{attribute 'qualified_only'}
{attribute 'to_string'}

TYPE eDataMappingVarNames :
(*
 * Enumeration for mapping every variable in ST_System_Monitor to a fixed
 * monitoring ID.  The hierarchy is fully expanded at every nesting level.
 *
 * Naming convention:
 *   Structs : <topLevel>_<field>_<subField>_..._<leafField>
 *   Arrays  : <path>_<indexName>  where the index names are:
 *               _AVG      (index 0)
 *               _L1       (index 1)
 *               _L2       (index 2)
 *               _L3       (index 3)
 *               _N        (index 4)
 *               _minimum  (index 5)
 *               _maximum  (index 6)
 *   Only electrical measurement arrays are individually expanded:
 *   ar_ActivePower, ar_ReactivePower, ar_ApparentPower,
 *   ar_PhaseVoltage, ar_LineVoltage, ar_Current,
 *   ar_Frequency, ar_THD, ar_PowerFactor.
 *   The aggregate array variable is NOT included; only individual
 *   per-index entries are present (e.g. ar_Current_AVG, ar_Current_L1).
 *
 *)
(	
None													:= 0,
	(*═════════════════════════════════════════════════════════*)
	(*  Safety and System State    *)
	(*═════════════════════════════════════════════════════════*)
	safety_b_SafetyOK                                          , (* BOOL *)
	safety_b_EstopChannelAOK                                   , (* BOOL *)
	safety_b_EstopChannelBOK                                   , (* BOOL *)
	safety_b_InsulationMonitorOK                               , (* BOOL *)
	safety_b_MRCDBOK                                           , (* BOOL *)
	safety_b_InverterDoorOK                                    , (* BOOL *)
	safety_b_ZptOK                                             , (* BOOL *)
	system_b_SMSnumberConfigured                               , (* BOOL *)
	system_b_CustomNameConfigured                              , (* BOOL *)
	system_s_SystemName                                        , (* STRING(20) *)
	system_b_TransportModePending                              , (* BOOL *)
	system_b_DehumModePending                                  , (* BOOL *)
	system_e_State                                             , (* eSystemState *)
	system_e_gridmode                                          , (* eGridmode *)
	system_e_UgridPowermode                                    , (* eUgridPowermode *)
	system_b_StartAllowed                                      , (* BOOL *)
	system_r_CurrentEfficiency                                 , (* REAL *)
	system_r_AvgEfficiency                                     , (* REAL *)
	system_r_RoundtripEfficiency                               , (* REAL *)
	system_DT_SystemTime                                       , (* DT *)
	system_PowerController_r_CurrentAct                        , (* REAL *)
	system_PowerController_r_Sact                              , (* REAL *)
	system_PowerController_r_PAct                              , (* REAL *)
	system_PowerController_r_QAct                              , (* REAL *)
	system_PowerController_r_PhaseVoltageAct                   , (* REAL *)
	system_PowerController_r_PFact                             , (* REAL *)
	system_PowerController_r_FeedInCurrentLimitActual          , (* REAL *)
	system_PowerController_r_SupplyInCurrentLimitActual        , (* REAL *)
	system_PowerController_b_ThrottlingActive                  , (* BOOL *)
	system_PowerController_ui_ThrottlingType                   , (* UINT *)
	system_PowerController_events_b_ReactivePIDError           , (* BOOL *)
	system_PowerController_events_b_ActivePIDError             , (* BOOL *)
	system_PowerController_events_b_FreqShiftPIDError          , (* BOOL *)
	system_GenGridController_b_active                          , (* BOOL *)
	system_GenGridController_b_faultActive                     , (* BOOL *)
	system_GenGridController_b_gensetHot                       , (* BOOL *)
	system_GenGridController_b_gensetStarting                  , (* BOOL *)
	system_GenGridController_b_ModeTransActive                 , (* BOOL *)
	system_GenGridController_b_ModeTransInhibit                , (* BOOL *)
	system_GenGridController_b_ModeChanged                     , (* BOOL *)
	system_GenGridController_b_ShowModeTrans                   , (* BOOL *)
	system_GenGridController_b_extGensetMode                   , (* BOOL *)
	system_GenGridController_b_gensetcontrol                   , (* BOOL *)
	system_GenGridController_e_BreakerMode                     , (* eBreakerOperationMode *)
	system_GenGridController_e_PowerControlMode                , (* ePowerControlMode *)
	system_GenGridController_e_GensetMode                      , (* eGensetMode *)
	system_GenGridController_e_GensetStartStop                 , (* eGensetStartStop *)
	system_GenGridController_e_state                           , (* eGenGridState *)
	system_GenGridController_e_RunCondition                    , (* eRunCondition *)
	system_GenGridController_events_b_InvalidGensetParameters  , (* BOOL *)
	system_GenGridController_events_b_RotationFieldFault       , (* BOOL *)
	system_GenGridController_events_b_CurrentLimitDisconnect   , (* BOOL *)
	system_GenGridController_events_b_CurrentLimitTrip         , (* BOOL *)
	system_GenGridController_events_b_EmstopDisconnect         , (* BOOL *)
	system_GenGridController_events_b_ShutdownDisconnect       , (* BOOL *)
	system_GenGridController_events_b_OverloadTrip             , (* BOOL *)
	system_GenGridController_events_b_OverFreqTrip             , (* BOOL *)
	system_GenGridController_events_b_UnderFreqTrip            , (* BOOL *)
	system_GenGridController_events_b_OverVoltTrip             , (* BOOL *)
	system_GenGridController_events_b_UnderVoltTrip            , (* BOOL *)
	system_GenGridController_events_b_ShutdownTimeOut          , (* BOOL *)
	system_GenGridController_events_b_SynchronisationFault     , (* BOOL *)
	system_GenGridController_events_b_StartupFault             , (* BOOL *)
	system_GenGridController_events_b_WarmupFault              , (* BOOL *)
	system_GenGridController_events_b_GenDownTrip              , (* BOOL *)
	system_GenGridController_events_b_GridLostTrip             , (* BOOL *)
	system_GenGridController_events_b_TransToGenIsoInhibit     , (* BOOL *)
	system_GenGridController_events_b_TransToGenDroopInhibit   , (* BOOL *)
	system_GenGridController_events_b_TransToGenFixInhibit     , (* BOOL *)
	system_GenGridController_events_b_TransFromInputGridAckRQ  , (* BOOL *)
	system_GenGridController_events_b_TransFromInputGenAckRQ   , (* BOOL *)
	system_GenGridController_events_b_StartingInhibit          , (* BOOL *)
	system_events_b_RestartRequiredMachineName                 , (* BOOL *)
	system_events_b_TimeUpdateFailed                           , (* BOOL *)

	(*═════════════════════════════════════════════════════════*)
	(*  Power Conversion Hardware    *)
	(*═════════════════════════════════════════════════════════*)
	powerstack_e_State                                         , (* eStatusPowerStack *)
	powerstack_e_PowerState                                    , (* ePowerstate *)
	powerstack_e_InverterMode                                  , (* eInverterModes *)
	powerstack_e_PowerMode                                     , (* ePowerModes *)
	powerstack_e_ThrottlingStatus                              , (* ePowerModuleThrottlingState *)
	powerstack_r_VoltageDroop                                  , (* REAL *)
	powerstack_r_FrequencyDroop                                , (* REAL *)
	powerstack_r_ACVoltageD7                                   , (* REAL *)
	powerstack_r_FrequencyD7                                   , (* REAL *)
	powerstack_r_ActivePower                                   , (* REAL *)
	powerstack_r_ReactivePower                                 , (* REAL *)
	powerstack_r_Pmin                                          , (* REAL *)
	powerstack_r_Pmax                                          , (* REAL *)
	powerstack_r_QMax                                          , (* REAL *)
	powerstack_r_QMin                                          , (* REAL *)
	powerstack_r_Smax                                          , (* REAL *)
	powerstack_r_ACcurrentLimit                                , (* REAL *)
	powerstack_r_ACcurrentLimitMax                             , (* REAL *)
	powerstack_r_PowerChangeRate                               , (* REAL *)
	powerstack_r_ApparentPower                                 , (* REAL *)
	powerstack_r_CosPhi                                        , (* REAL *)
	powerstack_r_AcCurrent                                     , (* REAL *)
	powerstack_r_DCPower                                       , (* REAL *)
	powerstack_r_DCVoltage                                     , (* REAL *)
	powerstack_r_DCcurrent                                     , (* REAL *)
	powerstack_r_ACVoltageSupply                               , (* REAL *)
	powerstack_r_FrequencySupply                               , (* REAL *)
	powerstack_r_LoadPercent                                   , (* REAL *)
	powerstack_r_RatedCurrent                                  , (* REAL *)
	powerstack_r_RatedPower                                    , (* REAL *)
	powerstack_r_OvercurrentValueAct                           , (* REAL *)
	powerstack_r_OvercurrentValueMax                           , (* REAL *)
	powerstack_r_ThrottlingValueAct                            , (* REAL *)
	powerstack_b_GridTied                                      , (* BOOL *)
	powerstack_b_GridCodeCheckActive                           , (* BOOL *)
	powerstack_b_GridCodeOK                                    , (* BOOL *)
	powerstack_b_GridACdetected                                , (* BOOL *)
	powerstack_b_InverterGridFormingMode                       , (* BOOL *)
	powerstack_b_ACDetected                                    , (* BOOL *)
	powerstack_b_DCDetected                                    , (* BOOL *)
	powerstack_b_InverterRunning                               , (* BOOL *)
	powerstack_b_StartedState                                  , (* BOOL *)
	powerstack_b_ControlEnabled                                , (* BOOL *)
	powerstack_b_EcomodeAvailable                              , (* BOOL *)
	powerstack_b_StartEnabled                                  , (* BOOL *)
	powerstack_r_MaxTemperature                                , (* REAL *)
	powerstack_t_ShiftHoldTimeRemaining                        , (* TIME *)
	powerstack_t_GridCodeReconnectTime                         , (* TIME *)
	powerstack_Events_b_CoolingDerating                        , (* BOOL *)
	powerstack_Events_b_PlimitShiftingActive                   , (* BOOL *)
	powerstack_Events_b_DCdeviationHigh                        , (* BOOL *)
	powerstack_Events_b_TemperatureWarning                     , (* BOOL *)
	powerstack_Events_b_OvercurrentWarning                     , (* BOOL *)
	powerstack_Events_b_UndervoltageWarning                    , (* BOOL *)
	powerstack_Events_b_OvervoltageWarning                     , (* BOOL *)
	powerstack_Events_b_TemperatureDeviationHigh               , (* BOOL *)
	powerstack_Events_b_PlimitShutdownWarning                  , (* BOOL *)
	powerstack_Events_b_MasterWarning                          , (* BOOL *)
	powerstack_Events_b_SlaveWarning                           , (* BOOL *)
	powerstack_Events_b_GridCodeWarning                        , (* BOOL *)
	powerstack_Events_b_UnderFreqFault                         , (* BOOL *)
	powerstack_Events_b_OverFreqFault                          , (* BOOL *)
	powerstack_Events_b_UnderVoltageFault                      , (* BOOL *)
	powerstack_Events_b_OverVoltageFault                       , (* BOOL *)
	powerstack_Events_b_OvercurrentFault                       , (* BOOL *)
	powerstack_Events_b_PlimitShutdown                         , (* BOOL *)
	powerstack_Events_b_TemperatureFault                       , (* BOOL *)
	powerstack_Events_b_MasterFault                            , (* BOOL *)
	powerstack_Events_b_SlaveFault                             , (* BOOL *)
	powerstack_Events_b_NetcontactorFault                      , (* BOOL *)
	powerstack_Events_b_startupTimeOut                         , (* BOOL *)
	powerstack_Events_b_ShutdownTimeOut                        , (* BOOL *)
	powerstack_Events_ui_shutdownRemainingTime                 , (* UINT *)
	powerstack_PowermoduleMaster_b_online                      , (* BOOL *)
	powerstack_PowermoduleMaster_r_ApparentPower               , (* REAL *)
	powerstack_PowermoduleMaster_r_ActivePower                 , (* REAL *)
	powerstack_PowermoduleMaster_r_ReactivePower               , (* REAL *)
	powerstack_PowermoduleMaster_r_ACVoltageD7                 , (* REAL *)
	powerstack_PowermoduleMaster_r_VoltageDroop                , (* REAL *)
	powerstack_PowermoduleMaster_r_ACVoltageSupply             , (* REAL *)
	powerstack_PowermoduleMaster_r_FrequencyD7                 , (* REAL *)
	powerstack_PowermoduleMaster_r_FrequencyDroop              , (* REAL *)
	powerstack_PowermoduleMaster_r_FrequencySupply             , (* REAL *)
	powerstack_PowermoduleMaster_r_CurrentUnbalance            , (* REAL *)
	powerstack_PowermoduleMaster_r_DCPower                     , (* REAL *)
	powerstack_PowermoduleMaster_r_DCVoltage                   , (* REAL *)
	powerstack_PowermoduleMaster_r_DCCurrent                   , (* REAL *)
	powerstack_PowermoduleMaster_r_ACCurrent                   , (* REAL *)
	powerstack_PowermoduleMaster_r_ActiveCurrent               , (* REAL *)
	powerstack_PowermoduleMaster_r_ReactiveCurrent             , (* REAL *)
	powerstack_PowermoduleMaster_r_LoadPercent                 , (* REAL *)
	powerstack_PowermoduleMaster_r_D7SyncError                 , (* REAL *)
	powerstack_PowermoduleMaster_r_Pmin                        , (* REAL *)
	powerstack_PowermoduleMaster_r_Pmax                        , (* REAL *)
	powerstack_PowermoduleMaster_r_QMax                        , (* REAL *)
	powerstack_PowermoduleMaster_r_Qmin                        , (* REAL *)
	powerstack_PowermoduleMaster_r_Pset                        , (* REAL *)
	powerstack_PowermoduleMaster_r_Qset                        , (* REAL *)
	powerstack_PowermoduleMaster_r_ACcurrentLimit              , (* REAL *)
	powerstack_PowermoduleMaster_r_OverCurrentValue            , (* REAL *)
	powerstack_PowermoduleMaster_r_ModulationIndex             , (* REAL *)
	powerstack_PowermoduleMaster_r_TemperatureInverter         , (* REAL *)
	powerstack_PowermoduleMaster_r_TemperatureGridChoke_1      , (* REAL *)
	powerstack_PowermoduleMaster_r_TemperatureGridChoke_2      , (* REAL *)
	powerstack_PowermoduleMaster_r_TemperatureGridChoke_3      , (* REAL *)
	powerstack_PowermoduleMaster_r_TemperatureCMChoke_1        , (* REAL *)
	powerstack_PowermoduleMaster_r_TemperatureCMChoke_2        , (* REAL *)
	powerstack_PowermoduleMaster_r_TemperatureCMChoke_3        , (* REAL *)
	powerstack_PowermoduleMaster_r_TemperatureCMChoke_4        , (* REAL *)
	powerstack_PowermoduleMaster_r_TemperatureMax              , (* REAL *)
	powerstack_PowermoduleMaster_w_TemperatureFaultWord        , (* WORD *)
	powerstack_PowermoduleMaster_w_OperationHours              , (* WORD *)
	powerstack_PowermoduleMaster_e_PowerMode                   , (* ePowerModes *)
	powerstack_PowermoduleMaster_e_InverterMode                , (* eInverterModes *)
	powerstack_PowermoduleMaster_e_Status                      , (* eStatusPowermodule *)
	powerstack_PowermoduleMaster_e_ThrottlingStatus            , (* ePowerModuleThrottlingState *)
	powerstack_PowermoduleMaster_ui_InverterCommStatus         , (* UINT *)
	powerstack_PowermoduleMaster_ui_BuscouplerCommStatus       , (* UINT *)
	powerstack_PowermoduleMaster_b_MccbTripOK                  , (* BOOL *)
	powerstack_PowermoduleMaster_b_MccbUvr24VdcOK              , (* BOOL *)
	powerstack_PowermoduleMaster_b_MccbFb                      , (* BOOL *)
	powerstack_PowermoduleMaster_b_FanFb                       , (* BOOL *)
	powerstack_PowermoduleMaster_b_DCcontactorFb               , (* BOOL *)
	powerstack_PowermoduleMaster_b_PrechargeContactor          , (* BOOL *)
	powerstack_PowermoduleMaster_b_LimiterActive               , (* BOOL *)
	powerstack_PowermoduleMaster_StatusWord_b_ReadyToDCCharge  , (* BOOL *)
	powerstack_PowermoduleMaster_StatusWord_b_ReadyToOperate   , (* BOOL *)
	powerstack_PowermoduleMaster_StatusWord_b_Running          , (* BOOL *)
	powerstack_PowermoduleMaster_StatusWord_b_Fault            , (* BOOL *)
	powerstack_PowermoduleMaster_StatusWord_b_RunEnabled       , (* BOOL *)
	powerstack_PowermoduleMaster_StatusWord_b_QuickstopNotActive, (* BOOL *)
	powerstack_PowermoduleMaster_StatusWord_b_MCCBControlNotOK , (* BOOL *)
	powerstack_PowermoduleMaster_StatusWord_b_Warning          , (* BOOL *)
	powerstack_PowermoduleMaster_StatusWord_b_DCAtReference    , (* BOOL *)
	powerstack_PowermoduleMaster_StatusWord_b_DCAboveLimit     , (* BOOL *)
	powerstack_PowermoduleMaster_StatusWord_b_WatchdogFeedback , (* BOOL *)
	powerstack_PowermoduleMaster_UgridStatusWord_b_ChargeControlActive, (* BOOL *)
	powerstack_PowermoduleMaster_UgridStatusWord_b_InternalChargingSwitchStatus, (* BOOL *)
	powerstack_PowermoduleMaster_UgridStatusWord_b_MCBcontrol  , (* BOOL *)
	powerstack_PowermoduleMaster_UgridStatusWord_b_MCBStatus   , (* BOOL *)
	powerstack_PowermoduleMaster_UgridStatusWord_b_RunEnabled  , (* BOOL *)
	powerstack_PowermoduleMaster_UgridStatusWord_b_DriveReady  , (* BOOL *)
	powerstack_PowermoduleMaster_UgridStatusWord_b_AFEmodeActive, (* BOOL *)
	powerstack_PowermoduleMaster_UgridStatusWord_b_IslandModeActive, (* BOOL *)
	powerstack_PowermoduleMaster_UgridStatusWord_b_MicrogridModeActive, (* BOOL *)
	powerstack_PowermoduleMaster_UgridStatusWord_b_RunRequestActive, (* BOOL *)
	powerstack_PowermoduleMaster_UgridStatusWord_b_DriveInRunState, (* BOOL *)
	powerstack_PowermoduleMaster_UgridStatusWord_b_FaultActive , (* BOOL *)
	powerstack_PowermoduleMaster_UgridStatusWord_b_SynchronizedToD7, (* BOOL *)
	powerstack_PowermoduleMaster_UgridStatusWord_b_D7MeasurementsOK, (* BOOL *)
	powerstack_PowermoduleMaster_GridcodeStatusWord_b_LineVoltTripLimHigh, (* BOOL *)
	powerstack_PowermoduleMaster_GridcodeStatusWord_b_LineVoltTripLimlow, (* BOOL *)
	powerstack_PowermoduleMaster_GridcodeStatusWord_b_LineFreqTripLimHigh, (* BOOL *)
	powerstack_PowermoduleMaster_GridcodeStatusWord_b_LineFreqTripLimLow, (* BOOL *)
	powerstack_PowermoduleMaster_GridcodeStatusWord_b_LineFreqOK, (* BOOL *)
	powerstack_PowermoduleMaster_GridcodeStatusWord_b_LineVoltOK, (* BOOL *)
	powerstack_PowermoduleMaster_GridcodeStatusWord_b_FRTActive, (* BOOL *)
	powerstack_PowermoduleMaster_GridcodeStatusWord_b_GridCodeTripActive, (* BOOL *)
	powerstack_PowermoduleMaster_Events_b_GeneralFaultFlag     , (* BOOL *)
	powerstack_PowermoduleMaster_Events_b_GeneralWarningFlag   , (* BOOL *)
	powerstack_PowermoduleMaster_Events_b_CMSTemperatureRangeWarning, (* BOOL *)
	powerstack_PowermoduleMaster_Events_b_FanStateUnknownWarning, (* BOOL *)
	powerstack_PowermoduleMaster_Events_b_TempThrottlingActive , (* BOOL *)
	powerstack_PowermoduleMaster_Events_b_CurrThrottlingActive , (* BOOL *)
	powerstack_PowermoduleMaster_Events_b_F1OverCurrent        , (* BOOL *)
	powerstack_PowermoduleMaster_Events_b_F2OverVoltage        , (* BOOL *)
	powerstack_PowermoduleMaster_Events_b_F9UnderVoltage       , (* BOOL *)
	powerstack_PowermoduleMaster_Events_b_F91ShortCircuit      , (* BOOL *)
	powerstack_PowermoduleMaster_Events_b_F3EarthFault         , (* BOOL *)
	powerstack_PowermoduleMaster_Events_b_Spare                , (* BOOL *)
	powerstack_PowermoduleMaster_Events_b_F14UnitOverTemperature, (* BOOL *)
	powerstack_PowermoduleMaster_Events_b_F56TemperatureFault  , (* BOOL *)
	powerstack_PowermoduleMaster_Events_b_F10LineSynchFault    , (* BOOL *)
	powerstack_PowermoduleMaster_Events_b_F52KeypadOCCommFault , (* BOOL *)
	powerstack_PowermoduleMaster_Events_b_F53FieldbusFault     , (* BOOL *)
	powerstack_PowermoduleMaster_Events_b_F59SystembusFault    , (* BOOL *)
	powerstack_PowermoduleMaster_Events_b_F54SlotCommunicationFault, (* BOOL *)
	powerstack_PowermoduleMaster_Events_b_F50Meas4mAFault      , (* BOOL *)
	powerstack_PowermoduleMaster_Events_b_F11OutputPhaseFault  , (* BOOL *)
	powerstack_PowermoduleMaster_Events_b_F80ChargeFault       , (* BOOL *)
	powerstack_PowermoduleMaster_Events_b_F51ExternalFault     , (* BOOL *)
	powerstack_PowermoduleMaster_Events_b_F31IGBTFault         , (* BOOL *)
	powerstack_PowermoduleMaster_Events_b_F64MCBstateFault     , (* BOOL *)
	powerstack_PowermoduleMaster_Events_b_WatchdogError        , (* BOOL *)
	powerstack_PowermoduleMaster_Events_b_24VdcUVRFault        , (* BOOL *)
	powerstack_PowermoduleMaster_Events_b_MCCBtrip             , (* BOOL *)
	powerstack_PowermoduleMaster_Events_b_ShutdownTimeOut      , (* BOOL *)
	powerstack_PowermoduleMaster_Events_b_StartUpTimeOut       , (* BOOL *)
	powerstack_PowermoduleMaster_Events_b_CMChokeTemperatureHigh_1  , (* BOOL *)
	powerstack_PowermoduleMaster_Events_b_CMChokeTemperatureHigh_2  , (* BOOL *)
	powerstack_PowermoduleMaster_Events_b_CMChokeTemperatureHigh_3  , (* BOOL *)
	powerstack_PowermoduleMaster_Events_b_CMChokeTemperatureHigh_4  , (* BOOL *)
	powerstack_PowermoduleMaster_Events_b_CMChokeTemperatureTooHigh_1  , (* BOOL *)
	powerstack_PowermoduleMaster_Events_b_CMChokeTemperatureTooHigh_2  , (* BOOL *)
	powerstack_PowermoduleMaster_Events_b_CMChokeTemperatureTooHigh_3  , (* BOOL *)
	powerstack_PowermoduleMaster_Events_b_CMChokeTemperatureTooHigh_4  , (* BOOL *)
	powerstack_PowermoduleMaster_Events_b_GridChokeTemperatureHigh_1  , (* BOOL *)
	powerstack_PowermoduleMaster_Events_b_GridChokeTemperatureHigh_2  , (* BOOL *)
	powerstack_PowermoduleMaster_Events_b_GridChokeTemperatureHigh_3  , (* BOOL *)
	powerstack_PowermoduleMaster_Events_b_GridChokeTemperatureTooHigh_1  , (* BOOL *)
	powerstack_PowermoduleMaster_Events_b_GridChokeTemperatureTooHigh_2  , (* BOOL *)
	powerstack_PowermoduleMaster_Events_b_GridChokeTemperatureTooHigh_3  , (* BOOL *)
	powerstack_PowermoduleMaster_Events_b_inverterTemperatureHigh, (* BOOL *)
	powerstack_PowermoduleMaster_Events_b_PT100Overrange       , (* BOOL *)
	powerstack_PowermoduleMaster_Events_b_PT100Underrange      , (* BOOL *)
	powerstack_PowermoduleMaster_Events_by_PT100ErrorCount     , (* BYTE *)
	powerstack_PowermoduleMaster_controldata_Controlword_b_ChargeDC, (* BOOL *)
	powerstack_PowermoduleMaster_controldata_Controlword_b_run , (* BOOL *)
	powerstack_PowermoduleMaster_controldata_Controlword_b_Reset, (* BOOL *)
	powerstack_PowermoduleMaster_controldata_Controlword_b_FieldbusControlEnable, (* BOOL *)
	powerstack_PowermoduleMaster_controldata_Controlword_b_WatchdogPulse, (* BOOL *)
	powerstack_PowermoduleMaster_controldata_Controlword_b_ParallelAFE, (* BOOL *)
	powerstack_PowermoduleMaster_controldata_Controlword_b_PIDenable, (* BOOL *)
	powerstack_PowermoduleMaster_controldata_Controlword_b_GridCodeEnable, (* BOOL *)
	powerstack_PowermoduleMaster_controldata_Controlword_b_ExtGridcodeTrip, (* BOOL *)
	powerstack_PowermoduleMaster_controldata_ui_ControlwordValue, (* UINT *)
	powerstack_PowermoduleMaster_controldata_i_invertermode    , (* INT *)
	powerstack_PowermoduleMaster_controldata_i_BaseCurrentRef  , (* INT *)
	powerstack_PowermoduleMaster_controldata_i_ReactiveCurrentRef, (* INT *)
	powerstack_PowermoduleMaster_controldata_i_FrequencyDroop  , (* INT *)
	powerstack_PowermoduleMaster_controldata_i_VoltageDroop    , (* INT *)
	powerstack_PowermoduleMaster_controldata_i_FrequencyDroopOffset, (* INT *)
	powerstack_PowermoduleMaster_controldata_i_VoltageCorrection, (* INT *)
	powerstack_PowermoduleMaster_controldata_i_BaseRefRampRate , (* INT *)
	powerstack_PowermoduleMaster_controldata_i_StartPowerMode  , (* INT *)
	powerstack_PowermoduleMaster_controldata_i_StartVoltageMode, (* INT *)
	powerstack_PowermoduleMaster_controldata_i_OutActCurrentLimit, (* INT *)
	powerstack_PowermoduleMaster_controldata_i_InActCurrentLimit, (* INT *)
	powerstack_PowermoduleMaster_controldata_i_DCVramprate     , (* INT *)
	powerstack_PowermoduleSlave_b_online                       , (* BOOL *)
	powerstack_PowermoduleSlave_r_ApparentPower                , (* REAL *)
	powerstack_PowermoduleSlave_r_ActivePower                  , (* REAL *)
	powerstack_PowermoduleSlave_r_ReactivePower                , (* REAL *)
	powerstack_PowermoduleSlave_r_ACVoltageD7                  , (* REAL *)
	powerstack_PowermoduleSlave_r_VoltageDroop                 , (* REAL *)
	powerstack_PowermoduleSlave_r_ACVoltageSupply              , (* REAL *)
	powerstack_PowermoduleSlave_r_FrequencyD7                  , (* REAL *)
	powerstack_PowermoduleSlave_r_FrequencyDroop               , (* REAL *)
	powerstack_PowermoduleSlave_r_FrequencySupply              , (* REAL *)
	powerstack_PowermoduleSlave_r_CurrentUnbalance             , (* REAL *)
	powerstack_PowermoduleSlave_r_DCPower                      , (* REAL *)
	powerstack_PowermoduleSlave_r_DCVoltage                    , (* REAL *)
	powerstack_PowermoduleSlave_r_DCCurrent                    , (* REAL *)
	powerstack_PowermoduleSlave_r_ACCurrent                    , (* REAL *)
	powerstack_PowermoduleSlave_r_ActiveCurrent                , (* REAL *)
	powerstack_PowermoduleSlave_r_ReactiveCurrent              , (* REAL *)
	powerstack_PowermoduleSlave_r_LoadPercent                  , (* REAL *)
	powerstack_PowermoduleSlave_r_D7SyncError                  , (* REAL *)
	powerstack_PowermoduleSlave_r_Pmin                         , (* REAL *)
	powerstack_PowermoduleSlave_r_Pmax                         , (* REAL *)
	powerstack_PowermoduleSlave_r_QMax                         , (* REAL *)
	powerstack_PowermoduleSlave_r_Qmin                         , (* REAL *)
	powerstack_PowermoduleSlave_r_Pset                         , (* REAL *)
	powerstack_PowermoduleSlave_r_Qset                         , (* REAL *)
	powerstack_PowermoduleSlave_r_ACcurrentLimit               , (* REAL *)
	powerstack_PowermoduleSlave_r_OverCurrentValue             , (* REAL *)
	powerstack_PowermoduleSlave_r_ModulationIndex              , (* REAL *)
	powerstack_PowermoduleSlave_r_TemperatureInverter          , (* REAL *)
	powerstack_PowermoduleSlave_r_TemperatureGridChoke_1       , (* REAL *)
	powerstack_PowermoduleSlave_r_TemperatureGridChoke_2       , (* REAL *)
	powerstack_PowermoduleSlave_r_TemperatureGridChoke_3       , (* REAL *)
	powerstack_PowermoduleSlave_r_TemperatureCMChoke_1         , (* REAL *)
	powerstack_PowermoduleSlave_r_TemperatureCMChoke_2         , (* REAL *)
	powerstack_PowermoduleSlave_r_TemperatureCMChoke_3         , (* REAL *)
	powerstack_PowermoduleSlave_r_TemperatureCMChoke_4         , (* REAL *)
	powerstack_PowermoduleSlave_r_TemperatureMax               , (* REAL *)
	powerstack_PowermoduleSlave_w_TemperatureFaultWord         , (* WORD *)
	powerstack_PowermoduleSlave_w_OperationHours               , (* WORD *)
	powerstack_PowermoduleSlave_e_PowerMode                    , (* ePowerModes *)
	powerstack_PowermoduleSlave_e_InverterMode                 , (* eInverterModes *)
	powerstack_PowermoduleSlave_e_Status                       , (* eStatusPowermodule *)
	powerstack_PowermoduleSlave_e_ThrottlingStatus             , (* ePowerModuleThrottlingState *)
	powerstack_PowermoduleSlave_ui_InverterCommStatus          , (* UINT *)
	powerstack_PowermoduleSlave_ui_BuscouplerCommStatus        , (* UINT *)
	powerstack_PowermoduleSlave_b_MccbTripOK                   , (* BOOL *)
	powerstack_PowermoduleSlave_b_MccbUvr24VdcOK               , (* BOOL *)
	powerstack_PowermoduleSlave_b_MccbFb                       , (* BOOL *)
	powerstack_PowermoduleSlave_b_FanFb                        , (* BOOL *)
	powerstack_PowermoduleSlave_b_DCcontactorFb                , (* BOOL *)
	powerstack_PowermoduleSlave_b_PrechargeContactor           , (* BOOL *)
	powerstack_PowermoduleSlave_b_LimiterActive                , (* BOOL *)
	powerstack_PowermoduleSlave_StatusWord_b_ReadyToDCCharge   , (* BOOL *)
	powerstack_PowermoduleSlave_StatusWord_b_ReadyToOperate    , (* BOOL *)
	powerstack_PowermoduleSlave_StatusWord_b_Running           , (* BOOL *)
	powerstack_PowermoduleSlave_StatusWord_b_Fault             , (* BOOL *)
	powerstack_PowermoduleSlave_StatusWord_b_RunEnabled        , (* BOOL *)
	powerstack_PowermoduleSlave_StatusWord_b_QuickstopNotActive, (* BOOL *)
	powerstack_PowermoduleSlave_StatusWord_b_MCCBControlNotOK  , (* BOOL *)
	powerstack_PowermoduleSlave_StatusWord_b_Warning           , (* BOOL *)
	powerstack_PowermoduleSlave_StatusWord_b_DCAtReference     , (* BOOL *)
	powerstack_PowermoduleSlave_StatusWord_b_DCAboveLimit      , (* BOOL *)
	powerstack_PowermoduleSlave_StatusWord_b_WatchdogFeedback  , (* BOOL *)
	powerstack_PowermoduleSlave_UgridStatusWord_b_ChargeControlActive, (* BOOL *)
	powerstack_PowermoduleSlave_UgridStatusWord_b_InternalChargingSwitchStatus, (* BOOL *)
	powerstack_PowermoduleSlave_UgridStatusWord_b_MCBcontrol   , (* BOOL *)
	powerstack_PowermoduleSlave_UgridStatusWord_b_MCBStatus    , (* BOOL *)
	powerstack_PowermoduleSlave_UgridStatusWord_b_RunEnabled   , (* BOOL *)
	powerstack_PowermoduleSlave_UgridStatusWord_b_DriveReady   , (* BOOL *)
	powerstack_PowermoduleSlave_UgridStatusWord_b_AFEmodeActive, (* BOOL *)
	powerstack_PowermoduleSlave_UgridStatusWord_b_IslandModeActive, (* BOOL *)
	powerstack_PowermoduleSlave_UgridStatusWord_b_MicrogridModeActive, (* BOOL *)
	powerstack_PowermoduleSlave_UgridStatusWord_b_RunRequestActive, (* BOOL *)
	powerstack_PowermoduleSlave_UgridStatusWord_b_DriveInRunState, (* BOOL *)
	powerstack_PowermoduleSlave_UgridStatusWord_b_FaultActive  , (* BOOL *)
	powerstack_PowermoduleSlave_UgridStatusWord_b_SynchronizedToD7, (* BOOL *)
	powerstack_PowermoduleSlave_UgridStatusWord_b_D7MeasurementsOK, (* BOOL *)
	powerstack_PowermoduleSlave_GridcodeStatusWord_b_LineVoltTripLimHigh, (* BOOL *)
	powerstack_PowermoduleSlave_GridcodeStatusWord_b_LineVoltTripLimlow, (* BOOL *)
	powerstack_PowermoduleSlave_GridcodeStatusWord_b_LineFreqTripLimHigh, (* BOOL *)
	powerstack_PowermoduleSlave_GridcodeStatusWord_b_LineFreqTripLimLow, (* BOOL *)
	powerstack_PowermoduleSlave_GridcodeStatusWord_b_LineFreqOK, (* BOOL *)
	powerstack_PowermoduleSlave_GridcodeStatusWord_b_LineVoltOK, (* BOOL *)
	powerstack_PowermoduleSlave_GridcodeStatusWord_b_FRTActive , (* BOOL *)
	powerstack_PowermoduleSlave_GridcodeStatusWord_b_GridCodeTripActive, (* BOOL *)
	powerstack_PowermoduleSlave_Events_b_GeneralFaultFlag      , (* BOOL *)
	powerstack_PowermoduleSlave_Events_b_GeneralWarningFlag    , (* BOOL *)
	powerstack_PowermoduleSlave_Events_b_CMSTemperatureRangeWarning, (* BOOL *)
	powerstack_PowermoduleSlave_Events_b_FanStateUnknownWarning, (* BOOL *)
	powerstack_PowermoduleSlave_Events_b_TempThrottlingActive  , (* BOOL *)
	powerstack_PowermoduleSlave_Events_b_CurrThrottlingActive  , (* BOOL *)
	powerstack_PowermoduleSlave_Events_b_F1OverCurrent         , (* BOOL *)
	powerstack_PowermoduleSlave_Events_b_F2OverVoltage         , (* BOOL *)
	powerstack_PowermoduleSlave_Events_b_F9UnderVoltage        , (* BOOL *)
	powerstack_PowermoduleSlave_Events_b_F91ShortCircuit       , (* BOOL *)
	powerstack_PowermoduleSlave_Events_b_F3EarthFault          , (* BOOL *)
	powerstack_PowermoduleSlave_Events_b_Spare                 , (* BOOL *)
	powerstack_PowermoduleSlave_Events_b_F14UnitOverTemperature, (* BOOL *)
	powerstack_PowermoduleSlave_Events_b_F56TemperatureFault   , (* BOOL *)
	powerstack_PowermoduleSlave_Events_b_F10LineSynchFault     , (* BOOL *)
	powerstack_PowermoduleSlave_Events_b_F52KeypadOCCommFault  , (* BOOL *)
	powerstack_PowermoduleSlave_Events_b_F53FieldbusFault      , (* BOOL *)
	powerstack_PowermoduleSlave_Events_b_F59SystembusFault     , (* BOOL *)
	powerstack_PowermoduleSlave_Events_b_F54SlotCommunicationFault, (* BOOL *)
	powerstack_PowermoduleSlave_Events_b_F50Meas4mAFault       , (* BOOL *)
	powerstack_PowermoduleSlave_Events_b_F11OutputPhaseFault   , (* BOOL *)
	powerstack_PowermoduleSlave_Events_b_F80ChargeFault        , (* BOOL *)
	powerstack_PowermoduleSlave_Events_b_F51ExternalFault      , (* BOOL *)
	powerstack_PowermoduleSlave_Events_b_F31IGBTFault          , (* BOOL *)
	powerstack_PowermoduleSlave_Events_b_F64MCBstateFault      , (* BOOL *)
	powerstack_PowermoduleSlave_Events_b_WatchdogError         , (* BOOL *)
	powerstack_PowermoduleSlave_Events_b_24VdcUVRFault         , (* BOOL *)
	powerstack_PowermoduleSlave_Events_b_MCCBtrip              , (* BOOL *)
	powerstack_PowermoduleSlave_Events_b_ShutdownTimeOut       , (* BOOL *)
	powerstack_PowermoduleSlave_Events_b_StartUpTimeOut        , (* BOOL *)
	powerstack_PowermoduleSlave_Events_b_CMChokeTemperatureHigh_1  , (* BOOL *)
	powerstack_PowermoduleSlave_Events_b_CMChokeTemperatureHigh_2  , (* BOOL *)
	powerstack_PowermoduleSlave_Events_b_CMChokeTemperatureHigh_3  , (* BOOL *)
	powerstack_PowermoduleSlave_Events_b_CMChokeTemperatureHigh_4  , (* BOOL *)
	powerstack_PowermoduleSlave_Events_b_CMChokeTemperatureTooHigh_1  , (* BOOL *)
	powerstack_PowermoduleSlave_Events_b_CMChokeTemperatureTooHigh_2  , (* BOOL *)
	powerstack_PowermoduleSlave_Events_b_CMChokeTemperatureTooHigh_3  , (* BOOL *)
	powerstack_PowermoduleSlave_Events_b_CMChokeTemperatureTooHigh_4  , (* BOOL *)
	powerstack_PowermoduleSlave_Events_b_GridChokeTemperatureHigh_1  , (* BOOL *)
	powerstack_PowermoduleSlave_Events_b_GridChokeTemperatureHigh_2  , (* BOOL *)
	powerstack_PowermoduleSlave_Events_b_GridChokeTemperatureHigh_3  , (* BOOL *)
	powerstack_PowermoduleSlave_Events_b_GridChokeTemperatureTooHigh_1  , (* BOOL *)
	powerstack_PowermoduleSlave_Events_b_GridChokeTemperatureTooHigh_2  , (* BOOL *)
	powerstack_PowermoduleSlave_Events_b_GridChokeTemperatureTooHigh_3  , (* BOOL *)
	powerstack_PowermoduleSlave_Events_b_inverterTemperatureHigh, (* BOOL *)
	powerstack_PowermoduleSlave_Events_b_PT100Overrange        , (* BOOL *)
	powerstack_PowermoduleSlave_Events_b_PT100Underrange       , (* BOOL *)
	powerstack_PowermoduleSlave_Events_by_PT100ErrorCount      , (* BYTE *)
	powerstack_PowermoduleSlave_controldata_Controlword_b_ChargeDC, (* BOOL *)
	powerstack_PowermoduleSlave_controldata_Controlword_b_run  , (* BOOL *)
	powerstack_PowermoduleSlave_controldata_Controlword_b_Reset, (* BOOL *)
	powerstack_PowermoduleSlave_controldata_Controlword_b_FieldbusControlEnable, (* BOOL *)
	powerstack_PowermoduleSlave_controldata_Controlword_b_WatchdogPulse, (* BOOL *)
	powerstack_PowermoduleSlave_controldata_Controlword_b_ParallelAFE, (* BOOL *)
	powerstack_PowermoduleSlave_controldata_Controlword_b_PIDenable, (* BOOL *)
	powerstack_PowermoduleSlave_controldata_Controlword_b_GridCodeEnable, (* BOOL *)
	powerstack_PowermoduleSlave_controldata_Controlword_b_ExtGridcodeTrip, (* BOOL *)
	powerstack_PowermoduleSlave_controldata_ui_ControlwordValue, (* UINT *)
	powerstack_PowermoduleSlave_controldata_i_invertermode     , (* INT *)
	powerstack_PowermoduleSlave_controldata_i_BaseCurrentRef   , (* INT *)
	powerstack_PowermoduleSlave_controldata_i_ReactiveCurrentRef, (* INT *)
	powerstack_PowermoduleSlave_controldata_i_FrequencyDroop   , (* INT *)
	powerstack_PowermoduleSlave_controldata_i_VoltageDroop     , (* INT *)
	powerstack_PowermoduleSlave_controldata_i_FrequencyDroopOffset, (* INT *)
	powerstack_PowermoduleSlave_controldata_i_VoltageCorrection, (* INT *)
	powerstack_PowermoduleSlave_controldata_i_BaseRefRampRate  , (* INT *)
	powerstack_PowermoduleSlave_controldata_i_StartPowerMode   , (* INT *)
	powerstack_PowermoduleSlave_controldata_i_StartVoltageMode , (* INT *)
	powerstack_PowermoduleSlave_controldata_i_OutActCurrentLimit, (* INT *)
	powerstack_PowermoduleSlave_controldata_i_InActCurrentLimit, (* INT *)
	powerstack_PowermoduleSlave_controldata_i_DCVramprate      , (* INT *)
	powerstack_Netcontactor_e_NetConState                      , (* eNetcontactorState *)
	powerstack_Netcontactor_b_SyncCloseCommand                 , (* BOOL *)
	powerstack_Netcontactor_b_NetConFb                         , (* BOOL *)
	powerstack_Netcontactor_b_NetcontRightFb                   , (* BOOL *)
	powerstack_Netcontactor_b_NetcontLeftFb                    , (* BOOL *)
	powerstack_Netcontactor_events_b_AMFEnabled                , (* BOOL *)
	powerstack_Netcontactor_events_b_ContactorRightFbFault     , (* BOOL *)
	powerstack_Netcontactor_events_b_ContactorLeftFbFault      , (* BOOL *)
	powerstack_Netcontactor_events_b_ContactorFbTimeout        , (* BOOL *)
	powerstack_Netcontactor_events_b_PhaseRotationFault        , (* BOOL *)
	powerstack_Netcontactor_events_b_IllegalLeftFieldSelected  , (* BOOL *)
	powermonitor_PQMeterReady                                  , (* BOOL *)
	powermonitor_InputField_ar_ApparentPower_AVG               , (* REAL *)
	powermonitor_InputField_ar_ApparentPower_L1                , (* REAL *)
	powermonitor_InputField_ar_ApparentPower_L2                , (* REAL *)
	powermonitor_InputField_ar_ApparentPower_L3                , (* REAL *)
	powermonitor_InputField_ar_ReactivePower_AVG               , (* REAL *)
	powermonitor_InputField_ar_ReactivePower_L1                , (* REAL *)
	powermonitor_InputField_ar_ReactivePower_L2                , (* REAL *)
	powermonitor_InputField_ar_ReactivePower_L3                , (* REAL *)
	powermonitor_InputField_ar_ActivePower_AVG                 , (* REAL *)
	powermonitor_InputField_ar_ActivePower_L1                  , (* REAL *)
	powermonitor_InputField_ar_ActivePower_L2                  , (* REAL *)
	powermonitor_InputField_ar_ActivePower_L3                  , (* REAL *)
	powermonitor_InputField_r_EnergyConsumed                   , (* REAL *)
	powermonitor_InputField_r_EnergySupplied                   , (* REAL *)
	powermonitor_InputField_ar_THD_AVG                         , (* REAL *)
	powermonitor_InputField_ar_THD_L1                          , (* REAL *)
	powermonitor_InputField_ar_THD_L2                          , (* REAL *)
	powermonitor_InputField_ar_THD_L3                          , (* REAL *)
	powermonitor_InputField_ar_PowerFactor_AVG                 , (* REAL *)
	powermonitor_InputField_ar_PowerFactor_L1                  , (* REAL *)
	powermonitor_InputField_ar_PowerFactor_L2                  , (* REAL *)
	powermonitor_InputField_ar_PowerFactor_L3                  , (* REAL *)
	powermonitor_InputField_ar_Current_AVG                     , (* REAL *)
	powermonitor_InputField_ar_Current_L1                      , (* REAL *)
	powermonitor_InputField_ar_Current_L2                      , (* REAL *)
	powermonitor_InputField_ar_Current_L3                      , (* REAL *)
	powermonitor_InputField_ar_Current_N                       , (* REAL *)
	powermonitor_InputField_r_CurrentUnbalance                 , (* REAL *)
	powermonitor_InputField_e_ACrotationStatus                 , (* eACRotationState *)
	powermonitor_InputField_ar_PhaseVoltage_AVG                , (* REAL *)
	powermonitor_InputField_ar_PhaseVoltage_L1                 , (* REAL *)
	powermonitor_InputField_ar_PhaseVoltage_L2                 , (* REAL *)
	powermonitor_InputField_ar_PhaseVoltage_L3                 , (* REAL *)
	powermonitor_InputField_ar_LineVoltage_AVG                 , (* REAL *)
	powermonitor_InputField_ar_LineVoltage_L1                  , (* REAL *)
	powermonitor_InputField_ar_LineVoltage_L2                  , (* REAL *)
	powermonitor_InputField_ar_LineVoltage_L3                  , (* REAL *)
	powermonitor_InputField_li_TimeVoltZeroCrossup             , (* LINT *)
	powermonitor_InputField_ar_Frequency_AVG                   , (* REAL *)
	powermonitor_InputField_ar_Frequency_L1                    , (* REAL *)
	powermonitor_InputField_ar_Frequency_L2                    , (* REAL *)
	powermonitor_InputField_ar_Frequency_L3                    , (* REAL *)
	powermonitor_InputField_r_VoltageUnbalance                 , (* REAL *)
	powermonitor_InputField_r_loadshare                        , (* REAL *)
	powermonitor_InputField_Powerlock_1_ar_ApparentPower_AVG    , (* REAL *)
	powermonitor_InputField_Powerlock_2_ar_ApparentPower_AVG    , (* REAL *)
	powermonitor_InputField_Powerlock_1_ar_ApparentPower_L1    , (* REAL *)
	powermonitor_InputField_Powerlock_2_ar_ApparentPower_L1    , (* REAL *)
	powermonitor_InputField_Powerlock_1_ar_ApparentPower_L2    , (* REAL *)
	powermonitor_InputField_Powerlock_2_ar_ApparentPower_L2    , (* REAL *)
	powermonitor_InputField_Powerlock_1_ar_ApparentPower_L3    , (* REAL *)
	powermonitor_InputField_Powerlock_2_ar_ApparentPower_L3    , (* REAL *)
	powermonitor_InputField_Powerlock_1_ar_ReactivePower_AVG    , (* REAL *)
	powermonitor_InputField_Powerlock_2_ar_ReactivePower_AVG    , (* REAL *)
	powermonitor_InputField_Powerlock_1_ar_ReactivePower_L1    , (* REAL *)
	powermonitor_InputField_Powerlock_2_ar_ReactivePower_L1    , (* REAL *)
	powermonitor_InputField_Powerlock_1_ar_ReactivePower_L2    , (* REAL *)
	powermonitor_InputField_Powerlock_2_ar_ReactivePower_L2    , (* REAL *)
	powermonitor_InputField_Powerlock_1_ar_ReactivePower_L3    , (* REAL *)
	powermonitor_InputField_Powerlock_2_ar_ReactivePower_L3    , (* REAL *)
	powermonitor_InputField_Powerlock_1_ar_ActivePower_AVG     , (* REAL *)
	powermonitor_InputField_Powerlock_2_ar_ActivePower_AVG     , (* REAL *)
	powermonitor_InputField_Powerlock_1_ar_ActivePower_L1      , (* REAL *)
	powermonitor_InputField_Powerlock_2_ar_ActivePower_L1      , (* REAL *)
	powermonitor_InputField_Powerlock_1_ar_ActivePower_L2      , (* REAL *)
	powermonitor_InputField_Powerlock_2_ar_ActivePower_L2      , (* REAL *)
	powermonitor_InputField_Powerlock_1_ar_ActivePower_L3      , (* REAL *)
	powermonitor_InputField_Powerlock_2_ar_ActivePower_L3      , (* REAL *)
	powermonitor_InputField_Powerlock_1_r_EnergyConsumed       , (* REAL *)
	powermonitor_InputField_Powerlock_2_r_EnergyConsumed       , (* REAL *)
	powermonitor_InputField_Powerlock_1_r_EnergySupplied       , (* REAL *)
	powermonitor_InputField_Powerlock_2_r_EnergySupplied       , (* REAL *)
	powermonitor_InputField_Powerlock_1_ar_THD_AVG             , (* REAL *)
	powermonitor_InputField_Powerlock_2_ar_THD_AVG             , (* REAL *)
	powermonitor_InputField_Powerlock_1_ar_THD_L1              , (* REAL *)
	powermonitor_InputField_Powerlock_2_ar_THD_L1              , (* REAL *)
	powermonitor_InputField_Powerlock_1_ar_THD_L2              , (* REAL *)
	powermonitor_InputField_Powerlock_2_ar_THD_L2              , (* REAL *)
	powermonitor_InputField_Powerlock_1_ar_THD_L3              , (* REAL *)
	powermonitor_InputField_Powerlock_2_ar_THD_L3              , (* REAL *)
	powermonitor_InputField_Powerlock_1_ar_PowerFactor_AVG     , (* REAL *)
	powermonitor_InputField_Powerlock_2_ar_PowerFactor_AVG     , (* REAL *)
	powermonitor_InputField_Powerlock_1_ar_PowerFactor_L1      , (* REAL *)
	powermonitor_InputField_Powerlock_2_ar_PowerFactor_L1      , (* REAL *)
	powermonitor_InputField_Powerlock_1_ar_PowerFactor_L2      , (* REAL *)
	powermonitor_InputField_Powerlock_2_ar_PowerFactor_L2      , (* REAL *)
	powermonitor_InputField_Powerlock_1_ar_PowerFactor_L3      , (* REAL *)
	powermonitor_InputField_Powerlock_2_ar_PowerFactor_L3      , (* REAL *)
	powermonitor_InputField_Powerlock_1_ar_Current_AVG         , (* REAL *)
	powermonitor_InputField_Powerlock_2_ar_Current_AVG         , (* REAL *)
	powermonitor_InputField_Powerlock_1_ar_Current_L1          , (* REAL *)
	powermonitor_InputField_Powerlock_2_ar_Current_L1          , (* REAL *)
	powermonitor_InputField_Powerlock_1_ar_Current_L2          , (* REAL *)
	powermonitor_InputField_Powerlock_2_ar_Current_L2          , (* REAL *)
	powermonitor_InputField_Powerlock_1_ar_Current_L3          , (* REAL *)
	powermonitor_InputField_Powerlock_2_ar_Current_L3          , (* REAL *)
	powermonitor_InputField_Powerlock_1_ar_Current_N           , (* REAL *)
	powermonitor_InputField_Powerlock_2_ar_Current_N           , (* REAL *)
	powermonitor_InputField_Powerlock_1_r_CurrentUnbalance     , (* REAL *)
	powermonitor_InputField_Powerlock_2_r_CurrentUnbalance     , (* REAL *)
	powermonitor_OutputField_ar_ApparentPower_AVG              , (* REAL *)
	powermonitor_OutputField_ar_ApparentPower_L1               , (* REAL *)
	powermonitor_OutputField_ar_ApparentPower_L2               , (* REAL *)
	powermonitor_OutputField_ar_ApparentPower_L3               , (* REAL *)
	powermonitor_OutputField_ar_ReactivePower_AVG              , (* REAL *)
	powermonitor_OutputField_ar_ReactivePower_L1               , (* REAL *)
	powermonitor_OutputField_ar_ReactivePower_L2               , (* REAL *)
	powermonitor_OutputField_ar_ReactivePower_L3               , (* REAL *)
	powermonitor_OutputField_ar_ActivePower_AVG                , (* REAL *)
	powermonitor_OutputField_ar_ActivePower_L1                 , (* REAL *)
	powermonitor_OutputField_ar_ActivePower_L2                 , (* REAL *)
	powermonitor_OutputField_ar_ActivePower_L3                 , (* REAL *)
	powermonitor_OutputField_r_EnergyConsumed                  , (* REAL *)
	powermonitor_OutputField_r_EnergySupplied                  , (* REAL *)
	powermonitor_OutputField_ar_THD_AVG                        , (* REAL *)
	powermonitor_OutputField_ar_THD_L1                         , (* REAL *)
	powermonitor_OutputField_ar_THD_L2                         , (* REAL *)
	powermonitor_OutputField_ar_THD_L3                         , (* REAL *)
	powermonitor_OutputField_ar_PowerFactor_AVG                , (* REAL *)
	powermonitor_OutputField_ar_PowerFactor_L1                 , (* REAL *)
	powermonitor_OutputField_ar_PowerFactor_L2                 , (* REAL *)
	powermonitor_OutputField_ar_PowerFactor_L3                 , (* REAL *)
	powermonitor_OutputField_ar_Current_AVG                    , (* REAL *)
	powermonitor_OutputField_ar_Current_L1                     , (* REAL *)
	powermonitor_OutputField_ar_Current_L2                     , (* REAL *)
	powermonitor_OutputField_ar_Current_L3                     , (* REAL *)
	powermonitor_OutputField_ar_Current_N                      , (* REAL *)
	powermonitor_OutputField_r_CurrentUnbalance                , (* REAL *)
	powermonitor_OutputField_e_ACrotationStatus                , (* eACRotationState *)
	powermonitor_OutputField_ar_PhaseVoltage_AVG               , (* REAL *)
	powermonitor_OutputField_ar_PhaseVoltage_L1                , (* REAL *)
	powermonitor_OutputField_ar_PhaseVoltage_L2                , (* REAL *)
	powermonitor_OutputField_ar_PhaseVoltage_L3                , (* REAL *)
	powermonitor_OutputField_ar_LineVoltage_AVG                , (* REAL *)
	powermonitor_OutputField_ar_LineVoltage_L1                 , (* REAL *)
	powermonitor_OutputField_ar_LineVoltage_L2                 , (* REAL *)
	powermonitor_OutputField_ar_LineVoltage_L3                 , (* REAL *)
	powermonitor_OutputField_li_TimeVoltZeroCrossup            , (* LINT *)
	powermonitor_OutputField_ar_Frequency_AVG                  , (* REAL *)
	powermonitor_OutputField_ar_Frequency_L1                   , (* REAL *)
	powermonitor_OutputField_ar_Frequency_L2                   , (* REAL *)
	powermonitor_OutputField_ar_Frequency_L3                   , (* REAL *)
	powermonitor_OutputField_r_VoltageUnbalance                , (* REAL *)
	powermonitor_OutputField_r_loadshare                       , (* REAL *)
	powermonitor_OutputField_Powerlock_1_ar_ApparentPower_AVG    , (* REAL *)
	powermonitor_OutputField_Powerlock_2_ar_ApparentPower_AVG    , (* REAL *)
	powermonitor_OutputField_Powerlock_3_ar_ApparentPower_AVG    , (* REAL *)
	powermonitor_OutputField_Powerlock_1_ar_ApparentPower_L1    , (* REAL *)
	powermonitor_OutputField_Powerlock_2_ar_ApparentPower_L1    , (* REAL *)
	powermonitor_OutputField_Powerlock_3_ar_ApparentPower_L1    , (* REAL *)
	powermonitor_OutputField_Powerlock_1_ar_ApparentPower_L2    , (* REAL *)
	powermonitor_OutputField_Powerlock_2_ar_ApparentPower_L2    , (* REAL *)
	powermonitor_OutputField_Powerlock_3_ar_ApparentPower_L2    , (* REAL *)
	powermonitor_OutputField_Powerlock_1_ar_ApparentPower_L3    , (* REAL *)
	powermonitor_OutputField_Powerlock_2_ar_ApparentPower_L3    , (* REAL *)
	powermonitor_OutputField_Powerlock_3_ar_ApparentPower_L3    , (* REAL *)
	powermonitor_OutputField_Powerlock_1_ar_ReactivePower_AVG    , (* REAL *)
	powermonitor_OutputField_Powerlock_2_ar_ReactivePower_AVG    , (* REAL *)
	powermonitor_OutputField_Powerlock_3_ar_ReactivePower_AVG    , (* REAL *)
	powermonitor_OutputField_Powerlock_1_ar_ReactivePower_L1    , (* REAL *)
	powermonitor_OutputField_Powerlock_2_ar_ReactivePower_L1    , (* REAL *)
	powermonitor_OutputField_Powerlock_3_ar_ReactivePower_L1    , (* REAL *)
	powermonitor_OutputField_Powerlock_1_ar_ReactivePower_L2    , (* REAL *)
	powermonitor_OutputField_Powerlock_2_ar_ReactivePower_L2    , (* REAL *)
	powermonitor_OutputField_Powerlock_3_ar_ReactivePower_L2    , (* REAL *)
	powermonitor_OutputField_Powerlock_1_ar_ReactivePower_L3    , (* REAL *)
	powermonitor_OutputField_Powerlock_2_ar_ReactivePower_L3    , (* REAL *)
	powermonitor_OutputField_Powerlock_3_ar_ReactivePower_L3    , (* REAL *)
	powermonitor_OutputField_Powerlock_1_ar_ActivePower_AVG    , (* REAL *)
	powermonitor_OutputField_Powerlock_2_ar_ActivePower_AVG    , (* REAL *)
	powermonitor_OutputField_Powerlock_3_ar_ActivePower_AVG    , (* REAL *)
	powermonitor_OutputField_Powerlock_1_ar_ActivePower_L1     , (* REAL *)
	powermonitor_OutputField_Powerlock_2_ar_ActivePower_L1     , (* REAL *)
	powermonitor_OutputField_Powerlock_3_ar_ActivePower_L1     , (* REAL *)
	powermonitor_OutputField_Powerlock_1_ar_ActivePower_L2     , (* REAL *)
	powermonitor_OutputField_Powerlock_2_ar_ActivePower_L2     , (* REAL *)
	powermonitor_OutputField_Powerlock_3_ar_ActivePower_L2     , (* REAL *)
	powermonitor_OutputField_Powerlock_1_ar_ActivePower_L3     , (* REAL *)
	powermonitor_OutputField_Powerlock_2_ar_ActivePower_L3     , (* REAL *)
	powermonitor_OutputField_Powerlock_3_ar_ActivePower_L3     , (* REAL *)
	powermonitor_OutputField_Powerlock_1_r_EnergyConsumed      , (* REAL *)
	powermonitor_OutputField_Powerlock_2_r_EnergyConsumed      , (* REAL *)
	powermonitor_OutputField_Powerlock_3_r_EnergyConsumed      , (* REAL *)
	powermonitor_OutputField_Powerlock_1_r_EnergySupplied      , (* REAL *)
	powermonitor_OutputField_Powerlock_2_r_EnergySupplied      , (* REAL *)
	powermonitor_OutputField_Powerlock_3_r_EnergySupplied      , (* REAL *)
	powermonitor_OutputField_Powerlock_1_ar_THD_AVG            , (* REAL *)
	powermonitor_OutputField_Powerlock_2_ar_THD_AVG            , (* REAL *)
	powermonitor_OutputField_Powerlock_3_ar_THD_AVG            , (* REAL *)
	powermonitor_OutputField_Powerlock_1_ar_THD_L1             , (* REAL *)
	powermonitor_OutputField_Powerlock_2_ar_THD_L1             , (* REAL *)
	powermonitor_OutputField_Powerlock_3_ar_THD_L1             , (* REAL *)
	powermonitor_OutputField_Powerlock_1_ar_THD_L2             , (* REAL *)
	powermonitor_OutputField_Powerlock_2_ar_THD_L2             , (* REAL *)
	powermonitor_OutputField_Powerlock_3_ar_THD_L2             , (* REAL *)
	powermonitor_OutputField_Powerlock_1_ar_THD_L3             , (* REAL *)
	powermonitor_OutputField_Powerlock_2_ar_THD_L3             , (* REAL *)
	powermonitor_OutputField_Powerlock_3_ar_THD_L3             , (* REAL *)
	powermonitor_OutputField_Powerlock_1_ar_PowerFactor_AVG    , (* REAL *)
	powermonitor_OutputField_Powerlock_2_ar_PowerFactor_AVG    , (* REAL *)
	powermonitor_OutputField_Powerlock_3_ar_PowerFactor_AVG    , (* REAL *)
	powermonitor_OutputField_Powerlock_1_ar_PowerFactor_L1     , (* REAL *)
	powermonitor_OutputField_Powerlock_2_ar_PowerFactor_L1     , (* REAL *)
	powermonitor_OutputField_Powerlock_3_ar_PowerFactor_L1     , (* REAL *)
	powermonitor_OutputField_Powerlock_1_ar_PowerFactor_L2     , (* REAL *)
	powermonitor_OutputField_Powerlock_2_ar_PowerFactor_L2     , (* REAL *)
	powermonitor_OutputField_Powerlock_3_ar_PowerFactor_L2     , (* REAL *)
	powermonitor_OutputField_Powerlock_1_ar_PowerFactor_L3     , (* REAL *)
	powermonitor_OutputField_Powerlock_2_ar_PowerFactor_L3     , (* REAL *)
	powermonitor_OutputField_Powerlock_3_ar_PowerFactor_L3     , (* REAL *)
	powermonitor_OutputField_Powerlock_1_ar_Current_AVG        , (* REAL *)
	powermonitor_OutputField_Powerlock_2_ar_Current_AVG        , (* REAL *)
	powermonitor_OutputField_Powerlock_3_ar_Current_AVG        , (* REAL *)
	powermonitor_OutputField_Powerlock_1_ar_Current_L1         , (* REAL *)
	powermonitor_OutputField_Powerlock_2_ar_Current_L1         , (* REAL *)
	powermonitor_OutputField_Powerlock_3_ar_Current_L1         , (* REAL *)
	powermonitor_OutputField_Powerlock_1_ar_Current_L2         , (* REAL *)
	powermonitor_OutputField_Powerlock_2_ar_Current_L2         , (* REAL *)
	powermonitor_OutputField_Powerlock_3_ar_Current_L2         , (* REAL *)
	powermonitor_OutputField_Powerlock_1_ar_Current_L3         , (* REAL *)
	powermonitor_OutputField_Powerlock_2_ar_Current_L3         , (* REAL *)
	powermonitor_OutputField_Powerlock_3_ar_Current_L3         , (* REAL *)
	powermonitor_OutputField_Powerlock_1_ar_Current_N          , (* REAL *)
	powermonitor_OutputField_Powerlock_2_ar_Current_N          , (* REAL *)
	powermonitor_OutputField_Powerlock_3_ar_Current_N          , (* REAL *)
	powermonitor_OutputField_Powerlock_1_r_CurrentUnbalance    , (* REAL *)
	powermonitor_OutputField_Powerlock_2_r_CurrentUnbalance    , (* REAL *)
	powermonitor_OutputField_Powerlock_3_r_CurrentUnbalance    , (* REAL *)
	powermonitor_InternalSupply_ar_ApparentPower_AVG           , (* REAL *)
	powermonitor_InternalSupply_ar_ApparentPower_L1            , (* REAL *)
	powermonitor_InternalSupply_ar_ApparentPower_L2            , (* REAL *)
	powermonitor_InternalSupply_ar_ApparentPower_L3            , (* REAL *)
	powermonitor_InternalSupply_ar_ReactivePower_AVG           , (* REAL *)
	powermonitor_InternalSupply_ar_ReactivePower_L1            , (* REAL *)
	powermonitor_InternalSupply_ar_ReactivePower_L2            , (* REAL *)
	powermonitor_InternalSupply_ar_ReactivePower_L3            , (* REAL *)
	powermonitor_InternalSupply_ar_ActivePower_AVG             , (* REAL *)
	powermonitor_InternalSupply_ar_ActivePower_L1              , (* REAL *)
	powermonitor_InternalSupply_ar_ActivePower_L2              , (* REAL *)
	powermonitor_InternalSupply_ar_ActivePower_L3              , (* REAL *)
	powermonitor_InternalSupply_r_EnergyConsumed               , (* REAL *)
	powermonitor_InternalSupply_r_EnergySupplied               , (* REAL *)
	powermonitor_InternalSupply_ar_THD_AVG                     , (* REAL *)
	powermonitor_InternalSupply_ar_THD_L1                      , (* REAL *)
	powermonitor_InternalSupply_ar_THD_L2                      , (* REAL *)
	powermonitor_InternalSupply_ar_THD_L3                      , (* REAL *)
	powermonitor_InternalSupply_ar_PowerFactor_AVG             , (* REAL *)
	powermonitor_InternalSupply_ar_PowerFactor_L1              , (* REAL *)
	powermonitor_InternalSupply_ar_PowerFactor_L2              , (* REAL *)
	powermonitor_InternalSupply_ar_PowerFactor_L3              , (* REAL *)
	powermonitor_InternalSupply_ar_Current_AVG                 , (* REAL *)
	powermonitor_InternalSupply_ar_Current_L1                  , (* REAL *)
	powermonitor_InternalSupply_ar_Current_L2                  , (* REAL *)
	powermonitor_InternalSupply_ar_Current_L3                  , (* REAL *)
	powermonitor_InternalSupply_ar_Current_N                   , (* REAL *)
	powermonitor_InternalSupply_r_CurrentUnbalance             , (* REAL *)
	powermonitor_BESS_e_ACrotationStatus                       , (* eACrotationState *)
	powermonitor_BESS_ar_Current_AVG                           , (* REAL *)
	powermonitor_BESS_ar_Current_L1                            , (* REAL *)
	powermonitor_BESS_ar_Current_L2                            , (* REAL *)
	powermonitor_BESS_ar_Current_L3                            , (* REAL *)
	powermonitor_BESS_ar_Current_N                             , (* REAL *)
	powermonitor_BESS_r_LineVoltage                            , (* REAL *)
	powermonitor_BESS_r_Frequency                              , (* REAL *)
	powermonitor_BESS_r_currentUnbalance                       , (* REAL *)
	powermonitor_BESS_r_ApparentPower                          , (* REAL *)
	powermonitor_BESS_r_ReactivePower                          , (* REAL *)
	powermonitor_BESS_r_ActivePower                            , (* REAL *)
	powermonitor_BESS_r_EnergyConsumed                         , (* REAL *)
	powermonitor_BESS_r_EnergySupplied                         , (* REAL *)
	powermonitor_BESS_r_PowerFactor                            , (* REAL *)
	powermonitor_events_b_MBCommWarning                        , (* BOOL *)
	powermonitor_events_b_MBCommError                          , (* BOOL *)
	powermonitor_events_b_MBTimeoutWarning                     , (* BOOL *)
	powermonitor_events_b_EL3443Warning                        , (* BOOL *)
	powermonitor_events_b_EL3443Error                          , (* BOOL *)
	powermonitor_events_b_ACdirectionDataInvalid               , (* BOOL *)
	ACswitchgear_b_InputSectionAvailable                       , (* BOOL *)
	ACswitchgear_b_InputMCCBfb                                 , (* BOOL *)
	ACswitchgear_b_InputMCCBShuntOK                            , (* BOOL *)
	ACswitchgear_b_OutputMCCBfb                                , (* BOOL *)
	ACswitchgear_b_OutputMCCBShuntOK                           , (* BOOL *)
	ACswitchgear_b_CEEprefuseOK                                , (* BOOL *)
	ACswitchgear_b_InputSynchronizerfb                         , (* BOOL *)
	ACswitchgear_b_InputContactorfb                            , (* BOOL *)
	ACswitchgear_b_PENlinkfb                                   , (* BOOL *)
	ACswitchgear_events_b_InputMCCBShuntFault                  , (* BOOL *)
	ACswitchgear_events_b_OutputMCCBShuntFault                 , (* BOOL *)
	ACswitchgear_events_b_CEEprefuseFault                      , (* BOOL *)
	ACswitchgear_events_b_InputContactorFault                  , (* BOOL *)
	neutraltransformer_b_active                                , (* BOOL *)
	neutraltransformer_r_TemperaturePhase_0                    , (* REAL *)
	neutraltransformer_r_TemperaturePhase_1                    , (* REAL *)
	neutraltransformer_r_TemperaturePhase_2                    , (* REAL *)
	neutraltransformer_r_TemperaturePhase_3                    , (* REAL *)
	neutraltransformer_r_TemperaturePhase_4                    , (* REAL *)
	neutraltransformer_r_TemperaturePhase_5                    , (* REAL *)
	neutraltransformer_r_TemperaturePhase_6                    , (* REAL *)
	neutraltransformer_r_Powerload                             , (* REAL *)
	neutraltransformer_r_ratedPower                            , (* REAL *)
	neutraltransformer_events_b_TemperatureHighPhase_1         , (* BOOL *)
	neutraltransformer_events_b_TemperatureHighPhase_2         , (* BOOL *)
	neutraltransformer_events_b_TemperatureHighPhase_3         , (* BOOL *)
	neutraltransformer_events_b_TemperatureTooHighPhase_1      , (* BOOL *)
	neutraltransformer_events_b_TemperatureTooHighPhase_2      , (* BOOL *)
	neutraltransformer_events_b_TemperatureTooHighPhase_3      , (* BOOL *)
	neutraltransformer_events_b_VoltageUnbalanceHigh           , (* BOOL *)
	neutraltransformer_events_b_VoltageUnbalanceTooHigh        , (* BOOL *)
	neutraltransformer_events_b_NeutralCurrentHigh             , (* BOOL *)
	neutraltransformer_events_b_NeutralCurrentTooHigh          , (* BOOL *)
	neutraltransformer_events_b_OvercurrentWarning             , (* BOOL *)
	neutraltransformer_events_b_OvercurrentAlarm               , (* BOOL *)
	DCswitchgear_b_couplingState                             	, (* BOOL *)
	DCswitchgear_r_Current                           			, (* REAL *)
	DCswitchgear_r_ratedCurrent                              	, (* REAL *)

	(*═════════════════════════════════════════════════════════*)
	(*  Energy Storage    *)
	(*═════════════════════════════════════════════════════════*)
	battery_BatteryInfo_b_BMSHeartBeatOK                       , (* BOOL *)
	battery_BatteryInfo_e_BMS_PowerOnStatus                    , (* ePowerOnStatus *)
	battery_BatteryInfo_e_BMS_Status                           , (* eBMS_Status *)
	battery_BatteryInfo_r_SystemVoltage                        , (* REAL *)
	battery_BatteryInfo_r_SystemCurrent                        , (* REAL *)
	battery_BatteryInfo_r_SOC                                  , (* REAL *)
	battery_BatteryInfo_r_SOH                                  , (* REAL *)
	battery_BatteryInfo_ar_CellVoltage_0                       , (* REAL *)
	battery_BatteryInfo_ar_CellVoltage_1                       , (* REAL *)
	battery_BatteryInfo_ar_CellVoltage_2                       , (* REAL *)
	battery_BatteryInfo_ar_CellTemperature_0                   , (* REAL *)
	battery_BatteryInfo_ar_CellTemperature_1                   , (* REAL *)
	battery_BatteryInfo_ar_CellTemperature_2                   , (* REAL *)
	battery_BatteryInfo_r_MaxChargeCurrentAllowed              , (* REAL *)
	battery_BatteryInfo_r_MaxDischargeCurrentAllowed           , (* REAL *)
	battery_BatteryInfo_r_MaxChargePowerAllowed                , (* REAL *)
	battery_BatteryInfo_r_MaxDischargePowerAllowed             , (* REAL *)
	battery_BatteryInfo_r_MaxSystemVoltageAllowed              , (* REAL *)
	battery_BatteryInfo_r_MinSystemVoltageAllowed              , (* REAL *)
	battery_BatteryInfo_r_SystemPower                          , (* REAL *)
	battery_BatteryInfo_r_ChargeSOE                            , (* REAL *)
	battery_BatteryInfo_r_DischargeSOE                         , (* REAL *)
	battery_BatteryInfo_r_RemainingChargeEnergy                , (* REAL *)
	battery_BatteryInfo_r_RemainingDischargeEnergy             , (* REAL *)
	battery_BatteryInfo_r_HistAccChargeEnergy                  , (* REAL *)
	battery_BatteryInfo_r_HistAccDischargeEnergy               , (* REAL *)
	battery_BatteryInfo_r_ratedPower                           , (* REAL *)
	battery_BatteryInfo_r_ratedCurrent                         , (* REAL *)
	battery_BatteryInfo_r_ratedEnergyCapacity                  , (* REAL *)
	battery_BatteryInfo_ui_CycleCount                          , (* UINT *)
	battery_BatteryInfo_r_SOCScaled                            , (* REAL *)
	battery_BatteryInfo_b_chargingAllowed                      , (* BOOL *)
	battery_BatteryInfo_b_dischargingAllowed                   , (* BOOL *)
	battery_BatteryInfo_r_RemainingDischargeEnergyNett         , (* REAL *)
	battery_BatteryInfo_r_RemainingChargeEnergyNett            , (* REAL *)
	battery_BatteryInfo_r_maxVoltageEver                       , (* REAL *)
	battery_BatteryInfo_r_maxChargeCurrentEver                 , (* REAL *)
	battery_BatteryInfo_r_maxDischargeCurrentEver              , (* REAL *)
	battery_T_RemainingTimeToAutoCalibration                   , (* TIME *)
	battery_MBMU_GeneralSBMUStatus_0                           , (* WORD *)
	battery_MBMU_GeneralSBMUStatus_1                           , (* WORD *)
	battery_MBMU_GeneralSBMUStatus_2                           , (* WORD *)
	battery_MBMU_GeneralSBMUStatus_3                           , (* WORD *)
	battery_MBMU_GeneralSBMUStatus_4                           , (* WORD *)
	battery_MBMU_GeneralSBMUStatus_5                           , (* WORD *)
	battery_MBMU_GeneralSBMUStatus_6                           , (* WORD *)
	battery_MBMU_GeneralSBMUStatus_7                           , (* WORD *)
	battery_MBMU_GeneralSBMUStatus_8                           , (* WORD *)
	battery_MBMU_GeneralSBMUStatus_9                           , (* WORD *)
	battery_MBMU_GeneralSBMUStatus_10                          , (* WORD *)
	battery_MBMU_GeneralSBMUStatus_11                          , (* WORD *)
	battery_MBMU_GeneralSBMUStatus_12                          , (* WORD *)
	battery_MBMU_GeneralSBMUStatus_13                          , (* WORD *)
	battery_MBMU_GeneralSBMUStatus_14                          , (* WORD *)
	battery_MBMU_GeneralSBMUStatus_15                          , (* WORD *)
	battery_MBMU_MBMUStatus_0                                  , (* WORD *)
	battery_MBMU_MBMUStatus_1                                  , (* WORD *)
	battery_MBMU_MBMUStatus_2                                  , (* WORD *)
	battery_MBMU_MBMUStatus_3                                  , (* WORD *)
	battery_MBMU_MBMUStatus_4                                  , (* WORD *)
	battery_MBMU_MBMUStatus_5                                  , (* WORD *)
	battery_MBMU_MBMUStatus_6                                  , (* WORD *)
	battery_MBMU_MBMUStatus_7                                  , (* WORD *)
	battery_MBMU_MBMUStatus_8                                  , (* WORD *)
	battery_MBMU_MBMUStatus_9                                  , (* WORD *)
	battery_MBMU_MBMUStatus_10                                 , (* WORD *)
	battery_MBMU_MBMUStatus_11                                 , (* WORD *)
	battery_MBMU_MBMUStatus_12                                 , (* WORD *)
	battery_MBMU_MBMUStatus_13                                 , (* WORD *)
	battery_MBMU_MBMUStatus_14                                 , (* WORD *)
	battery_MBMU_MBMUStatus_15                                 , (* WORD *)
	battery_MBMU_s_MBMU_SWVer                                  , (* STRING(16) *)
	battery_MBMU_s_MBMU_HWVer                                  , (* STRING(16) *)
	battery_MBMU_s_ETH_SWVer                                   , (* STRING(32) *)
	battery_MBMU_r_ETH_HWVer                                   , (* STRING(32) *)
	battery_MBMU_by_NumberOfSubSystems                         , (* BYTE *)
	battery_MBMU_DateTime_0                                    , (* WORD *)
	battery_MBMU_DateTime_1                                    , (* WORD *)
	battery_MBMU_DateTime_2                                    , (* WORD *)
	battery_MBMU_DateTime_3                                    , (* WORD *)
	battery_MBMU_DateTime_4                                    , (* WORD *)
	battery_MBMU_DateTime_5                                    , (* WORD *)
	battery_MBMU_b_InsulationSwitchOpen                        , (* BOOL *)
	battery_MBMU_BatteryStatus_b_BMSHeartBeatOK                , (* BOOL *)
	battery_MBMU_BatteryStatus_e_BMS_PowerOnStatus             , (* ePowerOnStatus *)
	battery_MBMU_BatteryStatus_e_BMS_Status                    , (* eBMS_Status *)
	battery_MBMU_BatteryStatus_r_SystemVoltage                 , (* REAL *)
	battery_MBMU_BatteryStatus_r_SystemCurrent                 , (* REAL *)
	battery_MBMU_BatteryStatus_r_SOC                           , (* REAL *)
	battery_MBMU_BatteryStatus_r_SOH                           , (* REAL *)
	battery_MBMU_BatteryStatus_ar_CellVoltage_0                , (* REAL *)
	battery_MBMU_BatteryStatus_ar_CellVoltage_1                , (* REAL *)
	battery_MBMU_BatteryStatus_ar_CellVoltage_2                , (* REAL *)
	battery_MBMU_BatteryStatus_ar_CellTemperature_0            , (* REAL *)
	battery_MBMU_BatteryStatus_ar_CellTemperature_1            , (* REAL *)
	battery_MBMU_BatteryStatus_ar_CellTemperature_2            , (* REAL *)
	battery_MBMU_BatteryStatus_r_MaxChargeCurrentAllowed       , (* REAL *)
	battery_MBMU_BatteryStatus_r_MaxDischargeCurrentAllowed    , (* REAL *)
	battery_MBMU_BatteryStatus_r_MaxChargePowerAllowed         , (* REAL *)
	battery_MBMU_BatteryStatus_r_MaxDischargePowerAllowed      , (* REAL *)
	battery_MBMU_BatteryStatus_r_MaxSystemVoltageAllowed       , (* REAL *)
	battery_MBMU_BatteryStatus_r_MinSystemVoltageAllowed       , (* REAL *)
	battery_MBMU_BatteryStatus_r_SystemPower                   , (* REAL *)
	battery_MBMU_BatteryStatus_r_ChargeSOE                     , (* REAL *)
	battery_MBMU_BatteryStatus_r_DischargeSOE                  , (* REAL *)
	battery_MBMU_BatteryStatus_r_RemainingChargeEnergy         , (* REAL *)
	battery_MBMU_BatteryStatus_r_RemainingDischargeEnergy      , (* REAL *)
	battery_MBMU_BatteryStatus_r_HistAccChargeEnergy           , (* REAL *)
	battery_MBMU_BatteryStatus_r_HistAccDischargeEnergy        , (* REAL *)
	battery_SBMU_0_w_SystemWarning                             , (* WORD *)
	battery_SBMU_1_w_SystemWarning                             , (* WORD *)
	battery_SBMU_2_w_SystemWarning                             , (* WORD *)
	battery_SBMU_3_w_SystemWarning                             , (* WORD *)
	battery_SBMU_0_SystemAlarm_0                               , (* WORD *)
	battery_SBMU_1_SystemAlarm_0                               , (* WORD *)
	battery_SBMU_2_SystemAlarm_0                               , (* WORD *)
	battery_SBMU_3_SystemAlarm_0                               , (* WORD *)
	battery_SBMU_0_SystemAlarm_1                               , (* WORD *)
	battery_SBMU_1_SystemAlarm_1                               , (* WORD *)
	battery_SBMU_2_SystemAlarm_1                               , (* WORD *)
	battery_SBMU_3_SystemAlarm_1                               , (* WORD *)
	battery_SBMU_0_SystemAlarm_2                               , (* WORD *)
	battery_SBMU_1_SystemAlarm_2                               , (* WORD *)
	battery_SBMU_2_SystemAlarm_2                               , (* WORD *)
	battery_SBMU_3_SystemAlarm_2                               , (* WORD *)
	battery_SBMU_0_b_PrechargeRelayClosed                      , (* BOOL *)
	battery_SBMU_1_b_PrechargeRelayClosed                      , (* BOOL *)
	battery_SBMU_2_b_PrechargeRelayClosed                      , (* BOOL *)
	battery_SBMU_3_b_PrechargeRelayClosed                      , (* BOOL *)
	battery_SBMU_0_b_MainPosRelayClosed                        , (* BOOL *)
	battery_SBMU_1_b_MainPosRelayClosed                        , (* BOOL *)
	battery_SBMU_2_b_MainPosRelayClosed                        , (* BOOL *)
	battery_SBMU_3_b_MainPosRelayClosed                        , (* BOOL *)
	battery_SBMU_0_b_MainNegRelayClosed                        , (* BOOL *)
	battery_SBMU_1_b_MainNegRelayClosed                        , (* BOOL *)
	battery_SBMU_2_b_MainNegRelayClosed                        , (* BOOL *)
	battery_SBMU_3_b_MainNegRelayClosed                        , (* BOOL *)
	battery_SBMU_0_b_ControlBoxFanOn                           , (* BOOL *)
	battery_SBMU_1_b_ControlBoxFanOn                           , (* BOOL *)
	battery_SBMU_2_b_ControlBoxFanOn                           , (* BOOL *)
	battery_SBMU_3_b_ControlBoxFanOn                           , (* BOOL *)
	battery_SBMU_0_b_BalanceStatus                             , (* BOOL *)
	battery_SBMU_1_b_BalanceStatus                             , (* BOOL *)
	battery_SBMU_2_b_BalanceStatus                             , (* BOOL *)
	battery_SBMU_3_b_BalanceStatus                             , (* BOOL *)
	battery_SBMU_0_b_DoorState                                 , (* BOOL *)
	battery_SBMU_1_b_DoorState                                 , (* BOOL *)
	battery_SBMU_2_b_DoorState                                 , (* BOOL *)
	battery_SBMU_3_b_DoorState                                 , (* BOOL *)
	battery_SBMU_0_s_SBMU_SWVer                                , (* STRING(16) *)
	battery_SBMU_1_s_SBMU_SWVer                                , (* STRING(16) *)
	battery_SBMU_2_s_SBMU_SWVer                                , (* STRING(16) *)
	battery_SBMU_3_s_SBMU_SWVer                                , (* STRING(16) *)
	battery_SBMU_0_s_SBMU_HWVer                                , (* STRING(16) *)
	battery_SBMU_1_s_SBMU_HWVer                                , (* STRING(16) *)
	battery_SBMU_2_s_SBMU_HWVer                                , (* STRING(16) *)
	battery_SBMU_3_s_SBMU_HWVer                                , (* STRING(16) *)
	battery_SBMU_0_s_CSC_SWVer                                 , (* STRING(16) *)
	battery_SBMU_1_s_CSC_SWVer                                 , (* STRING(16) *)
	battery_SBMU_2_s_CSC_SWVer                                 , (* STRING(16) *)
	battery_SBMU_3_s_CSC_SWVer                                 , (* STRING(16) *)
	battery_SBMU_0_s_CSC_HWVer                                 , (* STRING(16) *)
	battery_SBMU_1_s_CSC_HWVer                                 , (* STRING(16) *)
	battery_SBMU_2_s_CSC_HWVer                                 , (* STRING(16) *)
	battery_SBMU_3_s_CSC_HWVer                                 , (* STRING(16) *)
	battery_SBMU_0_BatteryStatus_r_SystemVoltage               , (* REAL *)
	battery_SBMU_1_BatteryStatus_r_SystemVoltage               , (* REAL *)
	battery_SBMU_2_BatteryStatus_r_SystemVoltage               , (* REAL *)
	battery_SBMU_3_BatteryStatus_r_SystemVoltage               , (* REAL *)
	battery_SBMU_0_BatteryStatus_r_SystemCurrent               , (* REAL *)
	battery_SBMU_1_BatteryStatus_r_SystemCurrent               , (* REAL *)
	battery_SBMU_2_BatteryStatus_r_SystemCurrent               , (* REAL *)
	battery_SBMU_3_BatteryStatus_r_SystemCurrent               , (* REAL *)
	battery_SBMU_0_BatteryStatus_r_SOC                         , (* REAL *)
	battery_SBMU_1_BatteryStatus_r_SOC                         , (* REAL *)
	battery_SBMU_2_BatteryStatus_r_SOC                         , (* REAL *)
	battery_SBMU_3_BatteryStatus_r_SOC                         , (* REAL *)
	battery_SBMU_0_BatteryStatus_r_SOH                         , (* REAL *)
	battery_SBMU_1_BatteryStatus_r_SOH                         , (* REAL *)
	battery_SBMU_2_BatteryStatus_r_SOH                         , (* REAL *)
	battery_SBMU_3_BatteryStatus_r_SOH                         , (* REAL *)
	battery_SBMU_0_BatteryStatus_ar_CellVoltage_0              , (* REAL *)
	battery_SBMU_1_BatteryStatus_ar_CellVoltage_0              , (* REAL *)
	battery_SBMU_2_BatteryStatus_ar_CellVoltage_0              , (* REAL *)
	battery_SBMU_3_BatteryStatus_ar_CellVoltage_0              , (* REAL *)
	battery_SBMU_0_BatteryStatus_ar_CellVoltage_1              , (* REAL *)
	battery_SBMU_1_BatteryStatus_ar_CellVoltage_1              , (* REAL *)
	battery_SBMU_2_BatteryStatus_ar_CellVoltage_1              , (* REAL *)
	battery_SBMU_3_BatteryStatus_ar_CellVoltage_1              , (* REAL *)
	battery_SBMU_0_BatteryStatus_ar_CellVoltage_2              , (* REAL *)
	battery_SBMU_1_BatteryStatus_ar_CellVoltage_2              , (* REAL *)
	battery_SBMU_2_BatteryStatus_ar_CellVoltage_2              , (* REAL *)
	battery_SBMU_3_BatteryStatus_ar_CellVoltage_2              , (* REAL *)
	battery_SBMU_0_BatteryStatus_ar_CellTemperature_0          , (* REAL *)
	battery_SBMU_1_BatteryStatus_ar_CellTemperature_0          , (* REAL *)
	battery_SBMU_2_BatteryStatus_ar_CellTemperature_0          , (* REAL *)
	battery_SBMU_3_BatteryStatus_ar_CellTemperature_0          , (* REAL *)
	battery_SBMU_0_BatteryStatus_ar_CellTemperature_1          , (* REAL *)
	battery_SBMU_1_BatteryStatus_ar_CellTemperature_1          , (* REAL *)
	battery_SBMU_2_BatteryStatus_ar_CellTemperature_1          , (* REAL *)
	battery_SBMU_3_BatteryStatus_ar_CellTemperature_1          , (* REAL *)
	battery_SBMU_0_BatteryStatus_ar_CellTemperature_2          , (* REAL *)
	battery_SBMU_1_BatteryStatus_ar_CellTemperature_2          , (* REAL *)
	battery_SBMU_2_BatteryStatus_ar_CellTemperature_2          , (* REAL *)
	battery_SBMU_3_BatteryStatus_ar_CellTemperature_2          , (* REAL *)
	battery_SBMU_0_BatteryStatus_r_MaxChargeCurrentAllowed     , (* REAL *)
	battery_SBMU_1_BatteryStatus_r_MaxChargeCurrentAllowed     , (* REAL *)
	battery_SBMU_2_BatteryStatus_r_MaxChargeCurrentAllowed     , (* REAL *)
	battery_SBMU_3_BatteryStatus_r_MaxChargeCurrentAllowed     , (* REAL *)
	battery_SBMU_0_BatteryStatus_r_MaxDischargeCurrentAllowed    , (* REAL *)
	battery_SBMU_1_BatteryStatus_r_MaxDischargeCurrentAllowed    , (* REAL *)
	battery_SBMU_2_BatteryStatus_r_MaxDischargeCurrentAllowed    , (* REAL *)
	battery_SBMU_3_BatteryStatus_r_MaxDischargeCurrentAllowed    , (* REAL *)
	battery_SBMU_0_BatteryStatus_r_HistAccChargeEnergy         , (* REAL *)
	battery_SBMU_1_BatteryStatus_r_HistAccChargeEnergy         , (* REAL *)
	battery_SBMU_2_BatteryStatus_r_HistAccChargeEnergy         , (* REAL *)
	battery_SBMU_3_BatteryStatus_r_HistAccChargeEnergy         , (* REAL *)
	battery_SBMU_0_BatteryStatus_r_HistAccDischargeEnergy      , (* REAL *)
	battery_SBMU_1_BatteryStatus_r_HistAccDischargeEnergy      , (* REAL *)
	battery_SBMU_2_BatteryStatus_r_HistAccDischargeEnergy      , (* REAL *)
	battery_SBMU_3_BatteryStatus_r_HistAccDischargeEnergy      , (* REAL *)
	battery_SBMU_0_BatteryStatus_w_MaxVoltageCellLocation      , (* WORD *)
	battery_SBMU_1_BatteryStatus_w_MaxVoltageCellLocation      , (* WORD *)
	battery_SBMU_2_BatteryStatus_w_MaxVoltageCellLocation      , (* WORD *)
	battery_SBMU_3_BatteryStatus_w_MaxVoltageCellLocation      , (* WORD *)
	battery_SBMU_0_BatteryStatus_w_MinVoltageCellLocation      , (* WORD *)
	battery_SBMU_1_BatteryStatus_w_MinVoltageCellLocation      , (* WORD *)
	battery_SBMU_2_BatteryStatus_w_MinVoltageCellLocation      , (* WORD *)
	battery_SBMU_3_BatteryStatus_w_MinVoltageCellLocation      , (* WORD *)
	battery_SBMU_0_BatteryStatus_w_MaxTempCellLocation         , (* WORD *)
	battery_SBMU_1_BatteryStatus_w_MaxTempCellLocation         , (* WORD *)
	battery_SBMU_2_BatteryStatus_w_MaxTempCellLocation         , (* WORD *)
	battery_SBMU_3_BatteryStatus_w_MaxTempCellLocation         , (* WORD *)
	battery_SBMU_0_BatteryStatus_w_MinTempCellLocation         , (* WORD *)
	battery_SBMU_1_BatteryStatus_w_MinTempCellLocation         , (* WORD *)
	battery_SBMU_2_BatteryStatus_w_MinTempCellLocation         , (* WORD *)
	battery_SBMU_3_BatteryStatus_w_MinTempCellLocation         , (* WORD *)
	battery_Events_b_COMMUNICATION_ERROR                       , (* BOOL *)
	battery_Events_b_OVER_TEMP_ALARM                           , (* BOOL *)
	battery_Events_b_OVER_TEMP_WARNING                         , (* BOOL *)
	battery_Events_b_UNDER_TEMP_ALARM                          , (* BOOL *)
	battery_Events_b_UNDER_TEMP_WARNING                        , (* BOOL *)
	battery_Events_b_OVER_CHARGE_CURRENT_ALARM                 , (* BOOL *)
	battery_Events_b_OVER_CHARGE_CURRENT_WARNING               , (* BOOL *)
	battery_Events_b_OVER_DISCHARGE_CURRENT_ALARM              , (* BOOL *)
	battery_Events_b_OVER_DISCHARGE_CURRENT_WARNING            , (* BOOL *)
	battery_Events_b_OVER_VOLT_ALARM                           , (* BOOL *)
	battery_Events_b_OVER_VOLT_WARNING                         , (* BOOL *)
	battery_Events_b_UNDER_VOLT_ALARM                          , (* BOOL *)
	battery_Events_b_UNDER_VOLT_WARNING                        , (* BOOL *)
	battery_Events_b_UNDER_SOC_MIN_ALARM                       , (* BOOL *)
	battery_Events_b_UNDER_SOC_MIN_WARNING                     , (* BOOL *)
	battery_Events_b_OVER_SOC_MAX_ALARM                        , (* BOOL *)
	battery_Events_b_OVER_SOC_MAX_WARNING                      , (* BOOL *)
	battery_Events_b_VOLTAGE_IMBALANCE_WARNING                 , (* BOOL *)
	battery_Events_b_TEMPERATURE_IMBALANCE_ALARM               , (* BOOL *)
	battery_Events_b_TEMPERATURE_IMBALANCE_WARNING             , (* BOOL *)
	battery_Events_b_CONTACTOR_ERROR                           , (* BOOL *)
	battery_Events_b_FAN_ERROR                                 , (* BOOL *)
	battery_Events_b_GROUND_FAULT                              , (* BOOL *)
	battery_Events_b_OPEN_DOOR_ERROR                           , (* BOOL *)
	battery_Events_b_CURRENT_IMBALANCE_WARNING                 , (* BOOL *)
	battery_Events_b_OTHER_ALARM                               , (* BOOL *)
	battery_Events_b_OTHER_WARNING                             , (* BOOL *)
	battery_Events_b_CONFIGURATION_ALARM                       , (* BOOL *)
	battery_Events_b_CONFIGURATION_WARNING                     , (* BOOL *)
	battery_Events_b_POWERONFAULT                              , (* BOOL *)
	battery_Events_b_POWEROFFFAULT                             , (* BOOL *)
	battery_Events_b_DISCONNECTOR_OFF                          , (* BOOL *)
	battery_Events_b_SocLowLimitOutOfRange                     , (* BOOL *)
	battery_Events_b_SocHighLimitOutOfRange                    , (* BOOL *)
	battery_Events_b_SBMUCommError_0                           , (* BOOL *)
	battery_Events_b_SBMUCommError_1                           , (* BOOL *)
	battery_Events_b_SBMUCommError_2                           , (* BOOL *)
	battery_Events_b_SBMUCommError_3                           , (* BOOL *)
	battery_Events_b_SBMUFailedToConnect_0                     , (* BOOL *)
	battery_Events_b_SBMUFailedToConnect_1                     , (* BOOL *)
	battery_Events_b_SBMUFailedToConnect_2                     , (* BOOL *)
	battery_Events_b_SBMUFailedToConnect_3                     , (* BOOL *)

	(*═════════════════════════════════════════════════════════*)
	(*  Protection Systems    *)
	(*═════════════════════════════════════════════════════════*)
	protections_FireDetection_b_FireAlarm                      , (* BOOL *)
	protections_FireDetection_SmokeDetectors_State             , (* eSmokeDetectAlarmStatus *)
	protections_FireDetection_CODetectors_State                , (* eCOAlarmStatus *)
	protections_FireDetection_CODetectors_b_CoValuesOK         , (* BOOL *)
	protections_FireDetection_CODetectors_Value_0              , (* REAL *)
	protections_FireDetection_CODetectors_Value_1              , (* REAL *)
	protections_FireDetection_CODetectors_Value_2              , (* REAL *)
	protections_FireDetection_CODetectors_Value_3              , (* REAL *)
	protections_FireDetection_Events_CODetFault                , (* BOOL *)
	protections_FireDetection_Events_CODetWarning1             , (* BOOL *)
	protections_FireDetection_Events_CODetWarning2             , (* BOOL *)
	protections_FireDetection_Events_CODetAlarm                , (* BOOL *)
	protections_FireDetection_Events_SmokeDetFault             , (* BOOL *)
	protections_FireDetection_Events_SmokeDetAlarm             , (* BOOL *)
	protections_FireDetection_Events_AlarmMuted                , (* BOOL *)
	protections_Insulation_b_Enabled                           , (* BOOL *)
	protections_Insulation_b_PENlinkDetected                   , (* BOOL *)
	protections_Insulation_b_Warning                           , (* BOOL *)
	protections_Insulation_e_EarthingSystemDetected            , (* eEarthingSystems *)
	protections_Insulation_b_PENlinkOperatedFault              , (* BOOL *)
	protections_Insulation_b_EarthingSystemMismatch            , (* BOOL *)
	protections_Insulation_b_NoEarthingSystemSet               , (* BOOL *)
	protections_MRCDB_b_prewarning                             , (* BOOL *)
	protections_Surge_b_Type12_OK                              , (* BOOL *)
	protections_Surge_b_Type3_OK                               , (* BOOL *)
	protections_OvercurrentProtection_r_TotalOutputCurrentLimit, (* REAL *)
	protections_OvercurrentProtection_r_TotalInputCurrentLimit , (* REAL *)
	protections_OvercurrentProtection_b_OutputWarning          , (* BOOL *)
	protections_OvercurrentProtection_b_InputWarning           , (* BOOL *)
	protections_OvercurrentProtection_b_OutputAlarm            , (* BOOL *)
	protections_OvercurrentProtection_b_InputAlarm             , (* BOOL *)
	protections_OvercurrentProtection_r_PeakCurrent            , (* REAL *)
	protections_OvercurrentProtection_t_PeakCurrentDuration    , (* TIME *)
	protections_OvercurrentProtection_s_locationPeak           , (* STRING *)
	peakshavebox_PSBmode                                       , (* ePSBMode *)
	peakshavebox_Powermonitor_ar_ApparentPower_AVG             , (* REAL *)
	peakshavebox_Powermonitor_ar_ApparentPower_L1              , (* REAL *)
	peakshavebox_Powermonitor_ar_ApparentPower_L2              , (* REAL *)
	peakshavebox_Powermonitor_ar_ApparentPower_L3              , (* REAL *)
	peakshavebox_Powermonitor_ar_ReactivePower_AVG             , (* REAL *)
	peakshavebox_Powermonitor_ar_ReactivePower_L1              , (* REAL *)
	peakshavebox_Powermonitor_ar_ReactivePower_L2              , (* REAL *)
	peakshavebox_Powermonitor_ar_ReactivePower_L3              , (* REAL *)
	peakshavebox_Powermonitor_ar_ActivePower_AVG               , (* REAL *)
	peakshavebox_Powermonitor_ar_ActivePower_L1                , (* REAL *)
	peakshavebox_Powermonitor_ar_ActivePower_L2                , (* REAL *)
	peakshavebox_Powermonitor_ar_ActivePower_L3                , (* REAL *)
	peakshavebox_Powermonitor_r_EnergyConsumed                 , (* REAL *)
	peakshavebox_Powermonitor_r_EnergySupplied                 , (* REAL *)
	peakshavebox_Powermonitor_ar_THD_AVG                       , (* REAL *)
	peakshavebox_Powermonitor_ar_THD_L1                        , (* REAL *)
	peakshavebox_Powermonitor_ar_THD_L2                        , (* REAL *)
	peakshavebox_Powermonitor_ar_THD_L3                        , (* REAL *)
	peakshavebox_Powermonitor_ar_PowerFactor_AVG               , (* REAL *)
	peakshavebox_Powermonitor_ar_PowerFactor_L1                , (* REAL *)
	peakshavebox_Powermonitor_ar_PowerFactor_L2                , (* REAL *)
	peakshavebox_Powermonitor_ar_PowerFactor_L3                , (* REAL *)
	peakshavebox_Powermonitor_ar_Current_AVG                   , (* REAL *)
	peakshavebox_Powermonitor_ar_Current_L1                    , (* REAL *)
	peakshavebox_Powermonitor_ar_Current_L2                    , (* REAL *)
	peakshavebox_Powermonitor_ar_Current_L3                    , (* REAL *)
	peakshavebox_Powermonitor_ar_Current_N                     , (* REAL *)
	peakshavebox_Powermonitor_r_CurrentUnbalance               , (* REAL *)
	peakshavebox_Powermonitor_e_ACrotationStatus               , (* eACRotationState *)
	peakshavebox_Powermonitor_ar_PhaseVoltage_AVG              , (* REAL *)
	peakshavebox_Powermonitor_ar_PhaseVoltage_L1               , (* REAL *)
	peakshavebox_Powermonitor_ar_PhaseVoltage_L2               , (* REAL *)
	peakshavebox_Powermonitor_ar_PhaseVoltage_L3               , (* REAL *)
	peakshavebox_Powermonitor_ar_LineVoltage_AVG               , (* REAL *)
	peakshavebox_Powermonitor_ar_LineVoltage_L1                , (* REAL *)
	peakshavebox_Powermonitor_ar_LineVoltage_L2                , (* REAL *)
	peakshavebox_Powermonitor_ar_LineVoltage_L3                , (* REAL *)
	peakshavebox_Powermonitor_li_TimeVoltZeroCrossup           , (* LINT *)
	peakshavebox_Powermonitor_ar_Frequency_AVG                 , (* REAL *)
	peakshavebox_Powermonitor_ar_Frequency_L1                  , (* REAL *)
	peakshavebox_Powermonitor_ar_Frequency_L2                  , (* REAL *)
	peakshavebox_Powermonitor_ar_Frequency_L3                  , (* REAL *)
	peakshavebox_Powermonitor_r_VoltageUnbalance               , (* REAL *)
	peakshavebox_PowerStatus_b_RotaryField                     , (* BOOL *)
	peakshavebox_PowerStatus_b_GeneralWarning                  , (* BOOL *)
	peakshavebox_PowerStatus_b_GeneralFault                    , (* BOOL *)
	peakshavebox_PowerStatus_b_OverVoltage                     , (* BOOL *)
	peakshavebox_PowerStatus_b_UnderVoltage                    , (* BOOL *)
	peakshavebox_PowerStatus_b_OverCurrent                     , (* BOOL *)
	peakshavebox_PowerStatus_b_Error_Phase_1                   , (* BOOL *)
	peakshavebox_PowerStatus_b_Error_Phase_2                   , (* BOOL *)
	peakshavebox_PowerStatus_b_Error_Phase_3                   , (* BOOL *)
	peakshavebox_r_MaxCTCurrent                                , (* REAL *)
	peakshavebox_b_buscouplerReady                             , (* BOOL *)
	peakshavebox_b_active                                      , (* BOOL *)
	peakshavebox_b_dataOK                                      , (* BOOL *)
	peakshavebox_b_ContactorFb                                 , (* BOOL *)
	peakshavebox_b_SyncFb                                      , (* BOOL *)
	peakshavebox_b_SettingsChangePending                       , (* BOOL *)

	(*═════════════════════════════════════════════════════════*)
	(*  Infrastructure and Auxiliary    *)
	(*═════════════════════════════════════════════════════════*)
	enclosure_climate_r_Humidity                               , (* REAL *)
	enclosure_climate_r_Temperature                            , (* REAL *)
	enclosure_climate_events_b_HumidityHigh                    , (* BOOL *)
	enclosure_climate_events_b_HumidityTooHigh                 , (* BOOL *)
	enclosure_climate_events_b_TemperatureHigh                 , (* BOOL *)
	enclosure_climate_events_b_TemperatureTooHigh              , (* BOOL *)
	enclosure_climate_events_b_TemperatureLow                  , (* BOOL *)
	enclosure_climate_events_b_TemperatureTooLow               , (* BOOL *)
	enclosure_climate_events_b_AIOverrange                     , (* BOOL *)
	enclosure_climate_events_b_AIUnderrange                    , (* BOOL *)
	enclosure_climate_events_b_AIError                         , (* BOOL *)
	enclosure_climate_events_b_DewpointTooHigh                 , (* BOOL *)
	enclosure_doors_b_ClientpanelDoorClosed                    , (* BOOL *)
	enclosure_doors_b_ControlPanelDoorClosed                   , (* BOOL *)
	enclosure_ledstrip_b_error                                 , (* BOOL *)
	enclosure_ledstrip_BeckhoffLed                             , (* BOOL *)
	internalpsu_b_24VdcAvailable                               , (* BOOL *)
	internalpsu_b_HVDCAvailable                                , (* BOOL *)
	internalpsu_b_400VACAvailable                              , (* BOOL *)
	internalpsu_e_400VSupplySource                             , (* e400VSupplySource *)
	internalpsu_UPS_r_InputVoltage                             , (* REAL *)
	internalpsu_UPS_r_OutputVoltage                            , (* REAL *)
	internalpsu_UPS_r_BatteryVoltage                           , (* REAL *)
	internalpsu_UPS_r_OutputCurrent                            , (* REAL *)
	internalpsu_UPS_ui_SOC                                     , (* UINT *)
	internalpsu_UPS_b_ChargerActive                            , (* BOOL *)
	internalpsu_UPS_b_SystemOnBattery                          , (* BOOL *)
	internalpsu_UPS_b_SystemOnDCInput                          , (* BOOL *)
	internalpsu_UPS_Events_b_BatteryLowInfo                    , (* BOOL *)
	internalpsu_UPS_Events_b_BatteryLowWarning                 , (* BOOL *)
	internalpsu_UPS_Events_b_BatteryLowError                   , (* BOOL *)
	internalpsu_UPS_Events_b_NoBatteryError                    , (* BOOL *)
	internalpsu_UPS_Events_b_InputVoltageWarning               , (* BOOL *)
	internalpsu_Events_b_DCPSUFault                            , (* BOOL *)
	internalpsu_Events_b_ACPSUFault                            , (* BOOL *)
	internalpsu_Events_b_GridInputFuseTripped                  , (* BOOL *)
	internalpsu_Events_b_CEEInputFuseTripped                   , (* BOOL *)
	internalpsu_Events_b_HVDCShutdownTimeExceeded              , (* BOOL *)
	internalpsu_Events_b_UPSLowShutdown                        , (* BOOL *)

